lrPowerPV_1 := fbPV.arrDataSymo10[1].lrPowerAcInverter;
lrPowerPV_2 := fbPV.arrDataSymo10[2].lrPowerAcInverter;
lrPowerPV_3 := fbPV.arrDataSymo10[3].lrPowerAcInverter;
lrPowerPV_4 := fbPV.arrDataSymo10[4].lrPowerAcInverter;
lrPowerPV_5 := fbPV.arrDataSymo10[5].lrPowerAcInverter;
lrPowerPV_6 := fbPV.arrDataSymo10[6].lrPowerAcInverter;
lrPowerPV_7 := fbPV.arrDataSymo10[7].lrPowerAcInverter;
lrPowerPV_8 := fbPV.arrDataSymo10[8].lrPowerAcInverter;

(*
fbPV_2.arrUnitID_Inverter[1] := 7;
fbPV_2.arrUnitID_Inverter[2] := 8;

fbPV_2(
	bEnable:= TRUE, 
	sIPAdress:= '192.168.10.4', 
	arrUnitID_Inverter:= , 
	arrDataSymo10=> , 
	stDataEMPower_PV=> , 
	stDataEMCounter_PV=> , 
	diNrOfEM_OUT_PV=> );

lrPowerPV_7 := fbPV_2.arrDataSymo10[1].lrPowerAcInverter;
lrPowerPV_8 := fbPV_2.arrDataSymo10[2].lrPowerAcInverter;

*)
	
fbPVInt(
	bEnable:= TRUE, 
	bPowerDataInvers:= , 
	diNrOfEM_IN_PV:= fbPV.diNrOfEM_OUT_PV, 
	stDataPv=> , 
	diNrOfPv_OUT=> );
	
lrPowerPV := lrPowerPV_1 + lrPowerPV_2 + lrPowerPV_3 + lrPowerPV_4 + lrPowerPV_5 + lrPowerPV_6 + lrPowerPV_7 + lrPowerPV_8;
byErrorWarningPV := fbPVInt.stDataPv.byErrorWarning;

// EnergyCounter
fbPVCounter(
	byActiveTariff:= 1, 
	lrPowerInput:= 0 - lrPowerPV, 
	lrTotalCounterEnergy_Consumption=> , 
	lrTotalCounterEnergy_Production=> , 
	lrCounterEnergyT1_Consumption=> , 
	lrCounterEnergyT2_Consumption=> , 
	lrCounterEnergyT1_Production=> , 
	lrCounterEnergyT2_Production=> );
	
IF fbPVCounter.lrTotalCounterEnergy_Production > lrCounterPV THEN  	
	lrCounterPV := fbPVCounter.lrTotalCounterEnergy_Production;
END_IF

END_PROGRAM

// ---- POUs/prgGrid.TcPOU
PROGRAM prgGrid
VAR PERSISTENT
	rSizeGridConn				: REAL;									//{#lynus.ag#()}
	lrCounterGridProd			: LREAL;								//{#lynus.ag#()}
	lrCounterGridCons			: LREAL;								//{#lynus.ag#()}
	lrCounterGridProd2			: LREAL;								//{#lynus.ag#()}
	lrCounterGridCons2			: LREAL;								//{#lynus.ag#()}
	r_kWh_PriceGridCons			: REAL;									//{#lynus.ag#()}
	r_kWh_PriceGridProd			: REAL;									//{#lynus.ag#()}
END_VAR
VAR
	fbGrid						: FB_Grid_Power;
	lrGridPower					: LREAL;								//{#lynus.ag#()}
	lrGridPower2				: LREAL;								//{#lynus.ag#()}
	lrGridPower2RealTime		: LREAL;								//{#lynus.ag#()}
	fbGridCounter				: FB_EnergyCounter;
	fbGrid2						: FB_Measurement_EL3413_v1;
END_VAR

fbGrid(
	bEnable:= TRUE, 
	diNrOfEMS_IN:= prgEMS.fbEMS.diNrOfEMS_OUT, 
	diNrOfEM_IN_Grid:= prgBattery.fbBattery.diNrOfEM_OUT_Grid, 
	rSizeGridConn:= rSizeGridConn, 
	stDataGrid=> , 
	diNrOfGrid_OUT=> );
	
lrGridPower := fbGrid.stDataGrid.lrPower;

// EnergyCounter
fbGridCounter(
	byActiveTariff:= 1, 
	lrPowerInput:= lrGridPower, 
	lrTotalCounterEnergy_Consumption=> , 
	lrTotalCounterEnergy_Production=> , 
	lrCounterEnergyT1_Consumption=> , 
	lrCounterEnergyT2_Consumption=> , 
	lrCounterEnergyT1_Production=> , 
	lrCounterEnergyT2_Production=> );
	
IF fbGridCounter.lrTotalCounterEnergy_Production > lrCounterGridProd THEN  	
	lrCounterGridProd := fbGridCounter.lrTotalCounterEnergy_Production;
END_IF

IF fbGridCounter.lrTotalCounterEnergy_Consumption > lrCounterGridCons THEN  	
	lrCounterGridCons := fbGridCounter.lrTotalCounterEnergy_Consumption;
END_IF

fbGrid2(
	bEnable:= true, 
	bInvers_CH1:= , 
	bInvers_CH2:= , 
	bInvers_CH3:= , 
	uiCurrentTransformerRatio:= 60, 
	stDataEMPower=> , 
	stDataEMCounter=> , 
	stDataEMPowerRealTime=> , 
	stDataEMCounterRealTime=> );
	
lrGridPower2 := fbGrid2.stDataEMPower.lrPowerTotal;
lrGridPower2RealTime := fbGrid2.stDataEMPowerRealTime.lrPowerTotal;
lrCounterGridProd2 := fbGrid2.stDataEMCounter.lrTotalCounterEnergy_Production;
lrCounterGridCons2 := fbGrid2.stDataEMCounter.lrTotalCounterEnergy_Consumption;

END_PROGRAM

// ---- FB/FB_Measurement_EL3413_v1.TcPOU
FUNCTION_BLOCK FB_Measurement_EL3413_v1
VAR_INPUT
	bEnable							: BOOL;											//Enable the function
 	bInvers_CH1						: BOOL;											//Invert the Output data from Channel 1 
	bInvers_CH2						: BOOL;											//Invert the Output data from Channel 2 
	bInvers_CH3						: BOOL;											//Invert the Output data from Channel 3
	uiCurrentTransformerRatio		: UINT;											//Current Transformer Ratio  
END_VAR
VAR_OUTPUT
	stDataEMPower					: ST_ElectricMeter_Output_Power;				//Output structure with Data from Electric Meter (Power Data) 
	stDataEMCounter					: ST_ElectricMeter_Output_Counter;				//Output structure with Data from Electric Meter (Counter Data) 
	stDataEMPowerRealTime			: ST_ElectricMeter_Output_Power;				//Output structure with Data from Electric Meter (Power Data RealTime)
	stDataEMCounterRealTime			: ST_ElectricMeter_Output_Counter;				//Output structure with Data from Electric Meter (Counter Data RealTime) 
	diNrOfEM_OUT					: DINT;											//Active Number from the Electric Meter for using on other functions

END_VAR
VAR
	structEL3413_IO : MDP5001_340_341_8D4302F4;
	timDissableFunctions			: TON;											//Timer to dissable the Function after Lynus_Standards.Constants_General.tTimeDissableLynusFunctions Days without connection to the Lynus Cloud
	timResetConnectionOnGVL			: TON;											//Timer to try reset the connection Flag on the GVL. (When somebody delete the Connection Function and make only a onlinechange)
	timSetCounterValues				: TON;											//Timer to set the counter values from the KL3403 Function to the EM Function
	real_Multiplier_CH1: REAL;
	real_Multiplier_CH2: REAL;
	real_Multiplier_CH3: REAL;
	fbEM							: FB_ElectricMeter;								//Electric Meter Function
	fbEnergyCounter					: FB_EnergyCounter;								//FB energy Counter, because the KL3403 has no nice logic for the Energy value
	fbNumberDevice					: FB_NumberOfDevice;							//Function block to calcualte the number of the Device
	iStateGVLData					: INT;											//State machine to handle the data on the GVL

	

	real_CT_sec1: REAL;
	real_f1_Hz: REAL;
	real_f2_Hz: REAL;
	real_f3_Hz: REAL;
	lreal_S_VA_L1: LREAL;
	lreal_S_VA_L2: LREAL;
	lreal_S_VA_L3: LREAL;
	lreal_Q_var_L1: LREAL;
	lreal_Q_var_L2: LREAL;
	lreal_Q_var_L3: LREAL;
	lreal_E1_kWh: LREAL;
	lreal_E2_kWh: LREAL;
	lreal_E3_kWh: LREAL;
END_VAR

//Creator : Stefan Lackner
//Company : EfficientIO
//Date : xx.09.2023
//Version : 1.0.0.0


//With this function is possible to read out all Information from a EL3443

//NOTE for diNr.....Designation => 
//_IN = Here Data come in from other Functions or go out to other functions about the GVL
//_OUT = Here Data go out to other functions about the GVL

(*-------------------------------------------------------------Calcualte the number of EM---------------------------------------------------------------*)

fbNumberDevice(
	diActualNumberOfDevices:= Lynus_Standards.GVL_Energy.stNumberOfDevices.diNumberOfElectricMeters, 
	diMaxNumberOfDevices:= Constants_Energy.diMaxNumberOfElectricMeters, 
	udiCounterOnlineChange:= TwinCAT_SystemInfoVarList._AppInfo.OnlineChangeCnt, 
	bNumberIsCalculatet=> , 
	bFPNumberIsCalculatet=> , 
	bOnlineChange=> , 
	diNumberForThisDevice=> diNrOfEM_OUT, 
	diNumberOfTotalDevices=> );

//Write new Numer on GVL
IF fbNumberDevice.bFPNumberIsCalculatet THEN
	Lynus_Standards.GVL_Energy.stNumberOfDevices.diNumberOfElectricMeters := fbNumberDevice.diNumberOfTotalDevices;	
END_IF

//Delete old Number on GVL
IF fbNumberDevice.bOnlineChange THEN 
	Lynus_Standards.GVL_Energy.stNumberOfDevices.diNumberOfElectricMeters := diNrOfEM_OUT;	
		iStateGVLData := 1; 
END_IF

(*-------------------------------------------------------------Service from Backend is ready and check the connection to backen for dissabel/enable Function---------------------------------------------------------------*)

//Try to reset the variable for connection on the GVL. When all is normal then the Lynus Mqtt connection function set this variable to true in the next cycle
//When we have no connection to the backend then after Lynus_Standards.Constants_General.tTimeDissableLynusFunctions days the Function is dissabled with all of his functionalities
timResetConnectionOnGVL(IN:= NOT timResetConnectionOnGVL.Q, PT:= T#1H, Q=> , ET=> );
IF timResetConnectionOnGVL.Q THEN 
	Lynus_Standards.GVL_Communicator.bStateConnectionToEnableFunctions := FALSE; 
END_IF
IF NOT Lynus_Standards.GVL_Communicator.bStateConnectionToEnableFunctions THEN 
	timDissableFunctions.IN := TRUE; 
ELSE 
	timDissableFunctions.IN := FALSE; 
END_IF  
timDissableFunctions(IN:= , PT:= Lynus_Standards.Constants_General.tTimeDissableLynusFunctions, Q=> , ET=> );

// limit inputs
uiCurrentTransformerRatio	 := LIMIT (1,uiCurrentTransformerRatio,10000);

//Invert the Output data, because it is possible that the current transformers have been mounted in different mounting positions.
IF NOT bInvers_CH1 THEN
	real_Multiplier_CH1 := 1;
ELSE
	real_Multiplier_CH1 := -1;
END_IF
IF NOT bInvers_CH2 THEN
	real_Multiplier_CH2 := 1;
ELSE
	real_Multiplier_CH2 := -1;
END_IF
IF NOT bInvers_CH3 THEN
	real_Multiplier_CH3 := 1;
ELSE
	real_Multiplier_CH3 := -1;
END_IF


//Function
fbEM(
	bEnable:= bEnable AND NOT timDissableFunctions.Q, 
	bError:= , 
	bEnableReadOutFunction:= FALSE, 
	bWriteWithDelay:= TRUE, 
	bPowerDataInvers:= FALSE,
	bReadOutDataDone:= timSetCounterValues.Q,
	iTimeReadOutInterval:= 0, 
	iErrorCode:= , 
	iWarningCode:= , 
	lrTotalCounterEnergy_Consumption:= fbEnergyCounter.lrTotalCounterEnergy_Consumption,
	lrTotalCounterEnergy_Production:= fbEnergyCounter.lrTotalCounterEnergy_Production, 
	lrCounterEnergyT1_Consumption:= fbEnergyCounter.lrCounterEnergyT1_Consumption,
	lrCounterEnergyT2_Consumption:= fbEnergyCounter.lrCounterEnergyT2_Consumption,
	lrCounterEnergyT1_Production:= fbEnergyCounter.lrCounterEnergyT1_Production, 
	lrCounterEnergyT2_Production:= fbEnergyCounter.lrCounterEnergyT2_Production, 
	lrCurrentL1:=  DINT_TO_LREAL(structEL3413_IO.MDP5001_340_341_Input.MDP5001_340_PM_Inputs_Channel_1_Current)/1000000 * uiCurrentTransformerRatio,
	lrVoltageL1N:= DINT_TO_LREAL(structEL3413_IO.MDP5001_340_341_Input.MDP5001_340_PM_Inputs_Channel_1_Voltage)/10000,
	lrVoltageL1L2:= fbEM.lrVoltageL1N * 1.73, 
	lrPowerL1:=  DINT_TO_LREAL(structEL3413_IO.MDP5001_340_341_Input.MDP5001_340_PM_Inputs_Channel_1_Active_power)/100 * uiCurrentTransformerRatio * real_Multiplier_CH1, 
	lrCurrentL2:=  DINT_TO_LREAL(structEL3413_IO.MDP5001_340_341_Input.MDP5001_340_PM_Inputs_Channel_2_Current)/1000000 * uiCurrentTransformerRatio,
	lrVoltageL2N:= DINT_TO_LREAL(structEL3413_IO.MDP5001_340_341_Input.MDP5001_340_PM_Inputs_Channel_2_Voltage)/10000,
	lrVoltageL2L3:= fbEM.lrVoltageL2N * 1.73,
	lrPowerL2:= DINT_TO_LREAL(structEL3413_IO.MDP5001_340_341_Input.MDP5001_340_PM_Inputs_Channel_2_Active_power)/100 * uiCurrentTransformerRatio * real_Multiplier_CH2,
	lrCurrentL3:=  DINT_TO_LREAL(structEL3413_IO.MDP5001_340_341_Input.MDP5001_340_PM_Inputs_Channel_3_Current)/1000000 * uiCurrentTransformerRatio,
	lrVoltageL3N:= DINT_TO_LREAL(structEL3413_IO.MDP5001_340_341_Input.MDP5001_340_PM_Inputs_Channel_3_Voltage)/10000,
	lrVoltageL3L1:= fbEM.lrVoltageL3N * 1.73,
	lrPowerL3:= DINT_TO_LREAL(structEL3413_IO.MDP5001_340_341_Input.MDP5001_340_PM_Inputs_Channel_3_Active_power)/100 * uiCurrentTransformerRatio * real_Multiplier_CH3,
	lrPowerTotal:= fbEM.lrPowerL1+fbEM.lrPowerL2+fbEM.lrPowerL3,
 	lrFrequency:= (real_f1_Hz + real_f2_Hz + real_f3_Hz)/3 , 
 	lrApparentPowerTotal:= (lreal_S_VA_L1 + lreal_S_VA_L2 + lreal_S_VA_L3),
	lrReactivePowerTotal:= (lreal_Q_var_L1 +lreal_Q_var_L2 + lreal_Q_var_L3), 
	tTimDelayOutput:= T#5S, 
	stDataEMOutPower=> stDataEMPowerRealTime, 
	stDataEMOutPowerDelay=> stDataEMPower, 
	stDataEMOutCounter=> stDataEMCounterRealTime,
	stDataEMOutCounterDelay=> stDataEMCounter,
	bReadOutMeter=> );
(*----------------------------------------------------------------------------------------Energy Counter Function----------------------------------------------------------------------------------------------*)

fbEnergyCounter(
	byActiveTariff:= 1, 
	lrPowerInput:= (fbEM.lrPowerTotal) / 1000, 
	lrTotalCounterEnergy_Consumption=> , 
	lrTotalCounterEnergy_Production=> , 
	lrCounterEnergyT1_Consumption=> , 
	lrCounterEnergyT2_Consumption=> , 
	lrCounterEnergyT1_Production=> , 
	lrCounterEnergyT2_Production=> );


IF (fbEM.lrPowerL1 * fbEM.lrPowerL1 + lreal_Q_var_L1 * lreal_Q_var_L1) <> 0 THEN 
	lreal_S_VA_L1:=SQRT(fbEM.lrPowerL1 * fbEM.lrPowerL1 + lreal_Q_var_L1 * lreal_Q_var_L1);
END_IF
IF (fbEM.lrPowerL2 * fbEM.lrPowerL2 + lreal_Q_var_L2 * lreal_Q_var_L2) <> 0 THEN 
	lreal_S_VA_L2:=SQRT(fbEM.lrPowerL2 * fbEM.lrPowerL2 + lreal_Q_var_L2 * lreal_Q_var_L2);
END_IF
IF (fbEM.lrPowerL3 * fbEM.lrPowerL3 + lreal_Q_var_L3 * lreal_Q_var_L3) <> 0 THEN 
	lreal_S_VA_L3:=SQRT(fbEM.lrPowerL3 * fbEM.lrPowerL3 + lreal_Q_var_L3 * lreal_Q_var_L3);
END_IF

CASE  structEL3413_IO.MDP5001_340_341_Input.MDP5001_340_PM_Inputs_Channel_1_Index OF
	1: (* Q *)
		lreal_Q_var_L1 :=DINT_TO_LREAL(structEL3413_IO.MDP5001_340_341_Input.MDP5001_340_PM_Inputs_Channel_1_Variant_value)/100 * uiCurrentTransformerRatio;
		structEL3413_IO.MDP5001_340_341_Output.MDP5001_340_PM_Outputs_Channel_1_Index := 2;
	2: (* E *)
		lreal_E1_kWh := DINT_TO_LREAL(structEL3413_IO.MDP5001_340_341_Input.MDP5001_340_PM_Inputs_Channel_1_Variant_value )/1000000 * uiCurrentTransformerRatio;
		structEL3413_IO.MDP5001_340_341_Output.MDP5001_340_PM_Outputs_Channel_1_Index := 4;
	4: (* f *)
		real_f1_Hz:=DINT_TO_REAL(structEL3413_IO.MDP5001_340_341_Input.MDP5001_340_PM_Inputs_Channel_1_Variant_value )/10;
		structEL3413_IO.MDP5001_340_341_Output.MDP5001_340_PM_Outputs_Channel_1_Index := 1;
ELSE
		structEL3413_IO.MDP5001_340_341_Output.MDP5001_340_PM_Outputs_Channel_1_Index := 1;
END_CASE
CASE  structEL3413_IO.MDP5001_340_341_Input.MDP5001_340_PM_Inputs_Channel_2_Index OF
	1: (* Q *)
		lreal_Q_var_L2 :=DINT_TO_LREAL(structEL3413_IO.MDP5001_340_341_Input.MDP5001_340_PM_Inputs_Channel_2_Variant_value)/100 * uiCurrentTransformerRatio;
		structEL3413_IO.MDP5001_340_341_Output.MDP5001_340_PM_Outputs_Channel_2_Index := 2;
	2: (* E *)
		lreal_E2_kWh := DINT_TO_LREAL(structEL3413_IO.MDP5001_340_341_Input.MDP5001_340_PM_Inputs_Channel_2_Variant_value )/1000000 * uiCurrentTransformerRatio;
		structEL3413_IO.MDP5001_340_341_Output.MDP5001_340_PM_Outputs_Channel_2_Index := 4;
	4: (* f *)
		real_f2_Hz:=DINT_TO_REAL(structEL3413_IO.MDP5001_340_341_Input.MDP5001_340_PM_Inputs_Channel_2_Variant_value )/10;
		structEL3413_IO.MDP5001_340_341_Output.MDP5001_340_PM_Outputs_Channel_2_Index := 1;
ELSE
		structEL3413_IO.MDP5001_340_341_Output.MDP5001_340_PM_Outputs_Channel_2_Index := 1;
END_CASE
CASE  structEL3413_IO.MDP5001_340_341_Input.MDP5001_340_PM_Inputs_Channel_3_Index OF
	1: (* Q *)
		lreal_Q_var_L3 :=DINT_TO_LREAL(structEL3413_IO.MDP5001_340_341_Input.MDP5001_340_PM_Inputs_Channel_3_Variant_value)/100 * uiCurrentTransformerRatio;
		structEL3413_IO.MDP5001_340_341_Output.MDP5001_340_PM_Outputs_Channel_3_Index := 2;
	2: (* E *)
		lreal_E3_kWh := DINT_TO_LREAL(structEL3413_IO.MDP5001_340_341_Input.MDP5001_340_PM_Inputs_Channel_3_Variant_value )/1000000 * uiCurrentTransformerRatio;
		structEL3413_IO.MDP5001_340_341_Output.MDP5001_340_PM_Outputs_Channel_3_Index := 4;
	4: (* f *)
		real_f3_Hz:=DINT_TO_REAL(structEL3413_IO.MDP5001_340_341_Input.MDP5001_340_PM_Inputs_Channel_3_Variant_value )/10;
		structEL3413_IO.MDP5001_340_341_Output.MDP5001_340_PM_Outputs_Channel_3_Index := 1;
ELSE
		structEL3413_IO.MDP5001_340_341_Output.MDP5001_340_PM_Outputs_Channel_3_Index := 1;
END_CASE


IF IsFinite(F_LREAL(fbEnergyCounter.lrTotalCounterEnergy_Production)) THEN stDataEMCounter.lrTotalCounterEnergy_Production := LINT_TO_LREAL(LREAL_TO_LINT(fbEnergyCounter.lrTotalCounterEnergy_Production * 100)) / 100; END_IF
IF IsFinite(F_LREAL(fbEnergyCounter.lrTotalCounterEnergy_Consumption)) THEN stDataEMCounter.lrTotalCounterEnergy_Consumption := LINT_TO_LREAL(LREAL_TO_LINT(fbEnergyCounter.lrTotalCounterEnergy_Consumption * 100)) / 100; END_IF

END_FUNCTION_BLOCK

// ---- POUs/prgCS.TcPOU
PROGRAM prgCS
VAR PERSISTENT
	bEnabledCS				: BOOL;									//{#lynus.ag#()}
	byPrioCS				: BYTE;									//{#lynus.ag#()}
	bySOC_E_CS				: BYTE;									//{#lynus.ag#()}
	bySOC_D_CS				: BYTE;									//{#lynus.ag#()}
	byMinPowerCS			: BYTE;									//{#lynus.ag#()}
	rMaxPowerCS				: REAL;									//{#lynus.ag#()}
	lrCounterCS				: LREAL;								//{#lynus.ag#()}
	bManualyOn				: BOOL;									//{#lynus.ag#()}
	byMinPower				: BYTE;									//{#lynus.ag#()}
	byManualyTargetPower	: BYTE;									//{#lynus.ag#()}
	m_ChargingLimit			: BOOL;									//{#lynus.ag#()}
	bOnEmergPowerOff		: BOOL;									//{#lynus.ag#()}
END_VAR
VAR
	fbCS					: FB_ECS_Alpitronic_Hypercharger_1;
	fbCSCounter				: FB_EnergyCounter;
	bIsEnabledCS			: BOOL;									//{#lynus.ag#()}
	byErrorWarningCS		: BYTE;									//{#lynus.ag#()}
	byStateMinPowerCS		: BYTE;									//{#lynus.ag#()}
	rTargetPowerCS			: REAL;									//{#lynus.ag#()}
	bCarConnected			: BOOL;									//{#lynus.ag#()}
	rChrgTime				: REAL;									//{#lynus.ag#()}
	lrPowerCS				: LREAL;								//{#lynus.ag#()}
	bSManualyOn				: BOOL;									//{#lynus.ag#()}
	bySManualyTargetPower	: BYTE;									//{#lynus.ag#()}
	str_IP: STRING(15):='192.168.10.10';
	rSOC_1					: REAL;									//{#lynus.ag#()}
	rSOC_2					: REAL;									//{#lynus.ag#()}
	f_Trig_CarConntected: f_trig;
	bSOnEmergPowerOff		: BOOL;									//{#lynus.ag#()}
END_VAR

fbCS.stSetupECS.byDisableSOC := bySOC_D_CS;
fbCS.stSetupECS.byEnableSOC := bySOC_E_CS;
fbCS.stSetupECS.byPriority := byPrioCS;
fbCS.stSetupECS.rMaxPower := rMaxPowerCS;
fbCS.stSetupECS.byCSMinPower := byMinPowerCS;
fbCS.stSetupECS.bManualyOn := bManualyOn;
fbCS.stSetupECS.byManualyTargetPower := byManualyTargetPower;
fbCS.stSetupECS.byCSMinPower := byMinPower;
fbCS.stSetupECS.bOnEmergPowerOff := bOnEmergPowerOff;


// Kofler special requirement for allowing to charge with maximium power and not PV surplus
// no battery used for charging the car. Battery Prio 2, CS prio 1
f_Trig_CarConntected(Clk := bCarConnected);
IF f_Trig_CarConntected.Q THEN 
	m_ChargingLimit := TRUE;
END_IF

IF m_ChargingLimit THEN
	fbCS.stSetupECS.byCSMinPower := byMinPowerCS;
ELSE
	fbCS.stSetupECS.byCSMinPower := 100;
END_IF
	
fbCS(
	bEnable:= bEnabledCS, 
	bPowerDataInvers:= , 
	byUnitID:= 1,				//Allways 1 
	diNrOfEMS_IN:= prgEMS.fbEMS.diNrOfEMS_OUT, 
	diNrOfEM_IN_CS:= , 
	sIPAdress:= str_IP, 
	stSetupECS:= , 
	stDataECS=> , 
	diNrOfECS_OUT=> );

bIsEnabledCS := fbCS.stDataECS.bEnabled;
byStateMinPowerCS := fbCS.stDataECS.bySCSMinPower;
rTargetPowerCS := fbCS.stDataECS.rTargetPower;	
byErrorWarningCS := fbCS.stDataECS.byErrorWarning;
bCarConnected := fbCS.stDataECS.bCarConnected;
rChrgTime := MAX(fbCS.stDataECS.arrChargingTimeInMin[1],fbCS.stDataECS.arrChargingTimeInMin[2]);
lrPowerCS := fbCS.stDataECS.lrTotalPower;
bSManualyOn := fbCS.stDataECS.bSManualyOn;
bSOnEmergPowerOff := fbCS.stDataECS.bSOnEmergPowerOff;

bySManualyTargetPower := fbCS.stDataECS.bySManualyTargetPower;
rSOC_1	:= DWORD_TO_REAL(fbCS.stDataECS.arrSocketSOCCar[1]);
rSOC_2	:= DWORD_TO_REAL(fbCS.stDataECS.arrSocketSOCCar[2]);						

// EnergyCounter
fbCSCounter(
	byActiveTariff:= 1, 
	lrPowerInput:= lrPowerCS, 
	lrTotalCounterEnergy_Consumption=> );
	
IF fbCSCounter.lrTotalCounterEnergy_Consumption > lrCounterCS THEN  	
	lrCounterCS := fbCSCounter.lrTotalCounterEnergy_Consumption;
END_IF

END_PROGRAM

// ---- FB/FB_ECS_Alpitronic_Hypercharger_1.TcPOU
FUNCTION_BLOCK FB_ECS_Alpitronic_Hypercharger_1
VAR_INPUT PERSISTENT
	bEnable										: BOOL;																			//{#lynus.ag#()} //Enable the Fuctionblock and his logic
	bPowerDataInvers							: BOOL;																			//With True its possible to invert all received power data from the electric meter
	byElectricFuseLine							: BYTE; 																		//Electric Fuse Line on wich the ECS is connected => 1 2 3 (If 0 then this charging station is not connected to a Electric Fuse Line)
	byUnitID									: BYTE;																			//Unit ID 
	diNrOfEMS_IN								: DINT;																			//Number of EMS what control this Device.
	diNrOfEM_IN_CS								: DINT;																			//Number of the electric meter for incoming power data. (Power Data for this Device)
	sIPAdress									: STRING(15);																	//IP Adress from the Alfen charging station
	stSetupECS									: ST_Setup_ECS;																	//{#lynus.ag#()} //Setup charging station
END_VAR
VAR_OUTPUT
	stDataECS									: ST_ECS_Output;																//{#lynus.ag#()} //Electric charging station output data
	diNrOfECS_OUT								: DINT;																			//Active Number from the Electric charging Function for using on other functions
	lrTotalPowerECSRealTime						: LREAL;																		//Total Electric Power in kW read out directly from the Charging station. (Real time)
END_VAR
VAR
	fbCS										: FB_ElectricChargingStation_1;													//Function block for electric charging station
	fbNumberDevice								: FB_NumberOfDevice;															//Function block to calcualte the number of the Device
	fbDIExternalLock							: FB_XL1XXX_DI;																	//Digital Input from external loock signal
	fbMBRead_FC4								: FB_MBReadInputRegs ;															//Modbus Read Function (FC4)
	fbMBWrite_FC16								: FB_MBWriteRegs;																//Modbus Write Function (FC16)
	fbConvertDwordToWord						: FB_CV_DWORD_TO_WORD;															//Convert Dword to Word
	fbConvertWordToDord							: FB_CV_WORD_TO_DWORD;															//Convert Word to Dword
	timDelay									: TON;																			//Timer for Delay between Requests
	timTimeout									: TON;																			//Timer for Timeout
	timDissableFunctions						: TON;																			//Timer to dissable the Function after Lynus_Standards.Constants_General.tTimeDissableLynusFunctions Days without connection to the Lynus Cloud
	timResetConnectionOnGVL						: TON;																			//Timer to try reset the connection Flag on the GVL. (When somebody delete the Connection Function and make only a onlinechange)
	timDelayStart								: TON;																			//Timer to start the state machine with Daley after enabling or after the system ist restartet
	FPError_FC_4								: R_TRIG;																		//Internal positive Edge
	FPError_FC_16								: R_TRIG;																		//Internal positive Edge
	FPEnable									: R_TRIG;																		//Internal positive Edge
	arrPD										: ARRAY[1..15] OF FB_PersistentData_Number;										//Function to save persistent data
	arrEnergyCounterSocket						: ARRAY[1..4] OF FB_EnergyCounter;												//FB energy Counter, because the charging station not deliver the total energy Counter in kWh
	fbPDString									: FB_PersistentData_String;														//Function to save persistent string data
	arrBuffer_FC4								: ARRAY[1..9] OF WORD;															//Buffer with Data from FC3
	arrBuffer_FC16								: ARRAY[1..2] OF WORD;															//Buffer with Data from FC16
	arrConnectorState							: ARRAY[1..4] OF WORD;															//Connector State
	arrChargingTime								: ARRAY[1..4] OF WORD;															//Charging Time in seconds
	arrSOCCar									: ARRAY[1..4] OF WORD;															//SOC from the Car
	arrPowerConnector							: ARRAY[1..4] OF DWORD;															//Power in W from each Connector
	arrEnergySession							: ARRAY[1..4] OF REAL;															//Energy Session in kWh
	bErrorCS									: BOOL;																			//Error State from the charging station
	bMBTCPError									: BOOL;																			//Modbus TCP Function Error																	
	byWaitInStep								: BYTE;																			//Wait in Step before start to clean data on PLC
	iStateGVLData								: INT;																			//State machine to handle the data on the GVL
	iStateModbusRead							: INT;																			//State machine for read out Data over Modbus RTU
	iStateModbusWrite							: INT;																			//State machine for write Data over Modbus RTU
	iStateModbusError							: INT;																			//State machine for error out Data over Modbus RTU	
	iStateModbus_CP								: INT;																			//Variable to compare the state machine variable to set or reset the timeout timer
	wNumberOfConnectors							: WORD;																			//Number of real connecotrs on the charging station
	wStationState								: WORD;																			//Charging Station State
	wConnectorInProgress						: WORD;																			//Shows the Connector in Progress when we have more then 1 Connector	
	diNumberOfActiveBatterys					: DINT;																			//Number of active batterys
	diNumberOfBatteryInverterInEPO				: DINT;																			//Number of battery inverters that work in Emergency Power operation 
	diLPForGVL									: DINT;																			//Loop to clean old data on GVL
	diCounterForGVL								: DINT;																			//Counter to clean old data on GVL
	dwSumSOC									: DWORD;																		//Sum of the SOC from all batterys
	dwTargetPower								: DWORD;																		//Target Power in Watt to send to the charging station
	liLPBatteryData								: LINT;																			//Loop to check some data from batterys
	liLPInEPO									: LINT;																			//Loop to check if 1 or more battery inverters build a island grid
	mtest: BOOL;

END_VAR
VAR PERSISTENT
	diNrOfEMS_IN_CP								: DINT;																			//Number of EMS what control this Device to compare with the original
END_VAR

//Creator : Kai Ebensperger
//Company : Lynus AG
//Date : 07.10.2021
//Version : 1.0.0.0

//With this Funcition its possible to communicate with a Alpitronic Hypercharger charging station over Modbus TCP.
//Its possible to controll the charging station over the charge power with the unit W
//This Charging station is a DC Hypercharger System.
//This API deliver the real Number of Connectors on the charging station
//To switch off the charging station send 0 Power to the charging station
//The minimal Curretn is set to 7.5 Ampere on AC site, bacause with al values that are < 5kW its not possible to charge the Car on DC site
//This Function Block support maximal 4 Connectors

//Versions that are supported : 1.3A Date : October 2020

//NOTE for diNr.....Designation => 
//_IN = Here Data come in from other Functions or go out to other functions about the GVL
//_OUT = Here Data go out to other functions about the GVL

(*--------------------------------------------------------------------------------------------Limits-------------------------------------------------------------------------------------*)

diNrOfEMS_IN := LIMIT(0,diNrOfEMS_IN,Constants_Energy.diMaxNumberOfEMS);
	diNrOfEM_IN_CS := LIMIT(0,diNrOfEM_IN_CS,Constants_Energy.diMaxNumberOfElectricMeters);	

(*------------------------------------------------------------------Power Data----------------------------------------------------------------------------*)

//Energy Counter Functions
arrEnergyCounterSocket[1](
	byActiveTariff:= 1, 
	lrPowerInput:= DWORD_TO_REAL(arrPowerConnector[1]) / 1000, 
	lrTotalCounterEnergy_Consumption=> , 
	lrTotalCounterEnergy_Production=> , 
	lrCounterEnergyT1_Consumption=> , 
	lrCounterEnergyT2_Consumption=> , 
	lrCounterEnergyT1_Production=> , 
	lrCounterEnergyT2_Production=> );
	
arrEnergyCounterSocket[2](
	byActiveTariff:= 1, 
	lrPowerInput:= DWORD_TO_REAL(arrPowerConnector[2]) / 1000, 
	lrTotalCounterEnergy_Consumption=> , 
	lrTotalCounterEnergy_Production=> , 
	lrCounterEnergyT1_Consumption=> , 
	lrCounterEnergyT2_Consumption=> , 
	lrCounterEnergyT1_Production=> , 
	lrCounterEnergyT2_Production=> );

arrEnergyCounterSocket[3](
	byActiveTariff:= 1, 
	lrPowerInput:= DWORD_TO_REAL(arrPowerConnector[3]) / 1000, 
	lrTotalCounterEnergy_Consumption=> , 
	lrTotalCounterEnergy_Production=> , 
	lrCounterEnergyT1_Consumption=> , 
	lrCounterEnergyT2_Consumption=> , 
	lrCounterEnergyT1_Production=> , 
	lrCounterEnergyT2_Production=> );	
	
arrEnergyCounterSocket[4](
	byActiveTariff:= 1, 
	lrPowerInput:= DWORD_TO_REAL(arrPowerConnector[4]) / 1000, 
	lrTotalCounterEnergy_Consumption=> , 
	lrTotalCounterEnergy_Production=> , 
	lrCounterEnergyT1_Consumption=> , 
	lrCounterEnergyT2_Consumption=> , 
	lrCounterEnergyT1_Production=> , 
	lrCounterEnergyT2_Production=> );

IF diNrOfEM_IN_CS <> 0 THEN
	//Energy Session Input data
	fbCS.bCalculateEnergySession := FALSE;
	fbCS.arrSocketPowerECS[1] := 0;
	fbCS.arrSocketPowerECS[2] := 0;
	fbCS.arrSocketPowerECS[3] := 0;
	fbCS.arrSocketPowerECS[4] := 0;
	fbCS.arrSocketEnergySession[1] := 0;
	fbCS.arrSocketEnergySession[2] := 0;
	fbCS.arrSocketEnergySession[3] := 0;
	fbCS.arrSocketEnergySession[4] := 0;
		IF NOT bPowerDataInvers THEN
			//Energy meter input data for cs Function block
			fbCS.lrCounterEnergyT1_Consumption := Lynus_Standards.GVL_Energy.stDataElectricMeters[diNrOfEM_IN_CS].lrCounterEnergyT1_Production * 1000;
			fbCS.lrCounterEnergyT2_Consumption := Lynus_Standards.GVL_Energy.stDataElectricMeters[diNrOfEM_IN_CS].lrCounterEnergyT2_Production * 1000;
			fbCS.lrCounterEnergyT1_Production := Lynus_Standards.GVL_Energy.stDataElectricMeters[diNrOfEM_IN_CS].lrCounterEnergyT1_Consumption * 1000;
			fbCS.lrCounterEnergyT2_Production := Lynus_Standards.GVL_Energy.stDataElectricMeters[diNrOfEM_IN_CS].lrCounterEnergyT1_Consumption * 1000;
			fbCS.lrTotalCounterEnergy_Consumption := Lynus_Standards.GVL_Energy.stDataElectricMeters[diNrOfEM_IN_CS].lrTotalCounterEnergy_Production * 1000;
			fbCS.lrTotalCounterEnergy_Production := Lynus_Standards.GVL_Energy.stDataElectricMeters[diNrOfEM_IN_CS].lrTotalCounterEnergy_Consumption * 1000;
				fbCS.lrTotalPowerECS := (Lynus_Standards.GVL_Energy.stDataElectricMeters[diNrOfEM_IN_CS].lrPower * 1000) * - 1;
		ELSE
			//Energy meter input data for cs Function block
			fbCS.lrCounterEnergyT1_Consumption := Lynus_Standards.GVL_Energy.stDataElectricMeters[diNrOfEM_IN_CS].lrCounterEnergyT1_Consumption * 1000;
			fbCS.lrCounterEnergyT2_Consumption := Lynus_Standards.GVL_Energy.stDataElectricMeters[diNrOfEM_IN_CS].lrCounterEnergyT2_Consumption * 1000;
			fbCS.lrCounterEnergyT1_Production := Lynus_Standards.GVL_Energy.stDataElectricMeters[diNrOfEM_IN_CS].lrCounterEnergyT1_Production * 1000;
			fbCS.lrCounterEnergyT2_Production := Lynus_Standards.GVL_Energy.stDataElectricMeters[diNrOfEM_IN_CS].lrCounterEnergyT2_Production * 1000;
			fbCS.lrTotalCounterEnergy_Consumption := Lynus_Standards.GVL_Energy.stDataElectricMeters[diNrOfEM_IN_CS].lrTotalCounterEnergy_Consumption * 1000;
			fbCS.lrTotalCounterEnergy_Production := Lynus_Standards.GVL_Energy.stDataElectricMeters[diNrOfEM_IN_CS].lrTotalCounterEnergy_Production * 1000;
				fbCS.lrTotalPowerECS := Lynus_Standards.GVL_Energy.stDataElectricMeters[diNrOfEM_IN_CS].lrPower * 1000;
		END_IF
ELSE
	//Energy meter input data for cs Function block
	fbCS.lrCounterEnergyT1_Consumption := arrEnergyCounterSocket[1].lrCounterEnergyT1_Consumption + arrEnergyCounterSocket[2].lrCounterEnergyT1_Consumption + arrEnergyCounterSocket[3].lrCounterEnergyT1_Consumption + arrEnergyCounterSocket[4].lrCounterEnergyT1_Consumption;
	fbCS.lrCounterEnergyT1_Consumption := fbCS.lrCounterEnergyT1_Consumption * 1000;
	fbCS.lrCounterEnergyT2_Consumption := arrEnergyCounterSocket[1].lrCounterEnergyT2_Consumption + arrEnergyCounterSocket[2].lrCounterEnergyT2_Consumption + arrEnergyCounterSocket[3].lrCounterEnergyT2_Consumption + arrEnergyCounterSocket[4].lrCounterEnergyT2_Consumption;
	fbCS.lrCounterEnergyT2_Consumption := fbCS.lrCounterEnergyT2_Consumption * 1000;
	fbCS.lrCounterEnergyT1_Production := arrEnergyCounterSocket[1].lrCounterEnergyT1_Production + arrEnergyCounterSocket[2].lrCounterEnergyT1_Production + arrEnergyCounterSocket[3].lrCounterEnergyT1_Production + arrEnergyCounterSocket[4].lrCounterEnergyT1_Production;
	fbCS.lrCounterEnergyT1_Production := fbCS.lrCounterEnergyT1_Production * 1000;
	fbCS.lrCounterEnergyT2_Production := arrEnergyCounterSocket[1].lrCounterEnergyT2_Production + arrEnergyCounterSocket[2].lrCounterEnergyT2_Production + arrEnergyCounterSocket[3].lrCounterEnergyT2_Production + arrEnergyCounterSocket[4].lrCounterEnergyT2_Production;
	fbCS.lrCounterEnergyT2_Production := fbCS.lrCounterEnergyT2_Production * 1000;
	fbCS.lrTotalCounterEnergy_Consumption := fbCS.lrCounterEnergyT1_Consumption + fbCS.lrCounterEnergyT2_Consumption;
	fbCS.lrTotalCounterEnergy_Production := fbCS.lrCounterEnergyT1_Production + fbCS.lrCounterEnergyT2_Production;
		fbCS.lrTotalPowerECS := arrPowerConnector[1] + arrPowerConnector[2] + arrPowerConnector[3] + arrPowerConnector[4];
	//Energy Session Input data
	fbCS.bCalculateEnergySession := FALSE;
	fbCS.arrSocketPowerECS[1] := arrPowerConnector[1];
	fbCS.arrSocketPowerECS[2] := arrPowerConnector[2];
	fbCS.arrSocketPowerECS[3] := arrPowerConnector[3];
	fbCS.arrSocketPowerECS[4] := arrPowerConnector[4];
	fbCS.arrSocketEnergySession[1] := arrEnergySession[1] * 1000;
	fbCS.arrSocketEnergySession[2] := arrEnergySession[2] * 1000;
	fbCS.arrSocketEnergySession[3] := arrEnergySession[3] * 1000;
	fbCS.arrSocketEnergySession[4] := arrEnergySession[4] * 1000;
END_IF			

(*-------------------------------------------------------------Calcualte the number of ECS---------------------------------------------------------------*)

fbNumberDevice(
	diActualNumberOfDevices:= Lynus_Standards.GVL_Energy.stNumberOfDevices.diNumberOfECS, 
	diMaxNumberOfDevices:= Constants_Energy.diMaxNumberOfElectricChargingStations, 
	udiCounterOnlineChange:= TwinCAT_SystemInfoVarList._AppInfo.OnlineChangeCnt, 
	bNumberIsCalculatet=> , 
	bFPNumberIsCalculatet=> , 
	bOnlineChange=> , 
	diNumberForThisDevice=> diNrOfECS_OUT, 
	diNumberOfTotalDevices=> );

//Write new Numer on GVL
IF fbNumberDevice.bFPNumberIsCalculatet THEN
	Lynus_Standards.GVL_Energy.stNumberOfDevices.diNumberOfECS := fbNumberDevice.diNumberOfTotalDevices;	
END_IF 

//Delete old Number on GVL
IF fbNumberDevice.bOnlineChange THEN 
	Lynus_Standards.GVL_Energy.stNumberOfDevices.diNumberOfECS := diNrOfECS_OUT;	
		iStateGVLData := 1;
END_IF

(*-------------------------------------------------------------Service from Backend is ready and check the connection to backen for dissabel/enable Function---------------------------------------------------------------*)

//Try to reset the variable for connection on the GVL. When all is normal then the Lynus Mqtt connection function set this variable to true in the next cycle
//When we have no connection to the backend then after Lynus_Standards.Constants_General.tTimeDissableLynusFunctions days the Function is dissabled with all of his functionalities
timResetConnectionOnGVL(IN:= NOT timResetConnectionOnGVL.Q, PT:= T#1H, Q=> , ET=> );
	IF timResetConnectionOnGVL.Q THEN Lynus_Standards.GVL_Communicator.bStateConnectionToEnableFunctions := FALSE; END_IF
		IF NOT Lynus_Standards.GVL_Communicator.bStateConnectionToEnableFunctions THEN timDissableFunctions.IN := TRUE; ELSE timDissableFunctions.IN := FALSE; END_IF  
			timDissableFunctions(IN:= , PT:= Lynus_Standards.Constants_General.tTimeDissableLynusFunctions, Q=> , ET=> );
			
(*--------------------------------------------------------------------------------------------State Machine Read--------------------------------------------------------------------------------------*)

//Timer for Delay
timDelay(IN:= , PT:= T#250MS, Q=> , ET=> );

//Timer for Timeout in Statemachine
IF (iStateModbusRead > 0 AND iStateModbusRead <= 3 AND iStateModbusRead = iStateModbus_CP) OR
		(iStateModbusWrite > 0 AND iStateModbusWrite <= 1 AND iStateModbusWrite = iStateModbus_CP) THEN
			timTimeout.IN := TRUE;
ELSE	
			timTimeout.IN := FALSE;
END_IF 
	//Timeout Timer is dissabled when the Init Step is aktiv or the function is not enabled
	IF (iStateModbusRead = 0 AND iStateModbusWrite = 0) OR NOT bEnable THEN timTimeout.IN := FALSE; END_IF
		timTimeout(IN:= , PT:= T#10S, Q=> , ET=> );

//Enable with Delay that not all sockets have to be created at the same time
timDelayStart(IN:= bEnable, PT:= T#20MS * diNrOfECS_OUT, Q=> , ET=> );
	FPEnable(CLK:= timDelayStart.Q, Q=> );

IF FPEnable.Q AND iStateModbusRead = 0 AND iStateModbusWrite = 0 THEN iStateModbusRead := 1; wConnectorInProgress := 1; END_IF		
		
//Not Enabled
IF NOT bEnable THEN iStateModbusRead := 0; iStateModbusError := 0; iStateModbusWrite := 0; END_IF		
		
CASE iStateModbusRead OF

	0://Init Step 
		iStateModbus_CP := 0;
			timDelay.IN := FALSE;
				fbMBRead_FC4.bExecute := FALSE;
					fbMBWrite_FC16.bExecute := FALSE;
						wConnectorInProgress := 0;
		arrConnectorState[1] := 0; arrConnectorState[2] := 0; arrConnectorState[3] := 0; arrConnectorState[4] := 0;
	
	1://Read Out the Number of connectors and the Charging station State (Register 2 and 3)
		iStateModbus_CP := iStateModbusRead;
		
		//Reset Write
		fbMBWrite_FC16.bExecute := FALSE;
			
		//Start Read
		fbMBRead_FC4.nQuantity := 2;
			fbMBRead_FC4.nMBAddr := 2;
				fbMBRead_FC4.bExecute := TRUE;
					fbMBRead_FC4.nUnitID := byUnitID;
			
		IF fbMBRead_FC4.bBusy THEN timDelay.IN := TRUE; END_IF
		
		//Wait for Delay, copy Data and then next step
		IF NOT fbMBRead_FC4.bBusy AND NOT fbMBRead_FC4.bError AND timDelay.Q THEN
			//Number of real Connectors
			wNumberOfConnectors := arrBuffer_FC4[1];
			//Charging station State
			wStationState := arrBuffer_FC4[2];	 
			//Connector in Progress
			wConnectorInProgress := LIMIT(1,wConnectorInProgress,4);
			//Go to Next Step
			fbMBRead_FC4.bExecute := FALSE;
				timDelay.IN := FALSE;		
					iStateModbusRead := 2;
		END_IF	

		//Error or Timeout
		IF FPError_FC_4.Q OR timTimeout.Q THEN
			iStateModbusError := 300;
		END_IF
		
	2://Read Out the Information of the real connecotrs (Register "1"00 to "1"08)
		iStateModbus_CP := iStateModbusRead;
		
		//Start Read
		fbMBRead_FC4.nQuantity := 9;
			fbMBRead_FC4.nMBAddr := 100 * wConnectorInProgress;
				fbMBRead_FC4.bExecute := TRUE;
					fbMBRead_FC4.nUnitID := byUnitID;
			
		IF fbMBRead_FC4.bBusy THEN timDelay.IN := TRUE; END_IF
		
		//Wait for Delay, copy Data and then next step
		IF NOT fbMBRead_FC4.bBusy AND NOT fbMBRead_FC4.bError AND timDelay.Q THEN
			//Connecotor State
			arrConnectorState[wConnectorInProgress] := arrBuffer_FC4[1];
			//Connector Power
			fbConvertWordToDord(wInputValue_1:= arrBuffer_FC4[5], wInputValue_2:= arrBuffer_FC4[6], eByteOrderForConvert:= eByteOrder.eBigEndian, dwOutputValue=> );
				arrPowerConnector[wConnectorInProgress] := fbConvertWordToDord.dwOutputValue;
			//Charging Time in Seconds
			arrChargingTime[wConnectorInProgress] := arrBuffer_FC4[7];
			//Energy Session
			arrEnergySession[wConnectorInProgress] := WORD_TO_REAL(arrBuffer_FC4[8]) / 100;
			//SOC from the Car
			arrSOCCar[wConnectorInProgress] := arrBuffer_FC4[9] / 100;
			//Go to Next Step
			fbMBRead_FC4.bExecute := FALSE;
				timDelay.IN := FALSE;		
					iStateModbusRead := 3;
		END_IF	

		//Error or Timeout
		IF FPError_FC_4.Q OR timTimeout.Q THEN
			iStateModbusError := 300;
		END_IF
		
	3://Wait 1 Step to reset the delay counter befor start to write
		iStateModbus_CP := iStateModbusRead;
		
			iStateModbusWrite := 1;
				//-1 because 0 is the Init Step for Read
				iStateModbusRead := - 1;
				
			//Error on Master, changes on Inputs or Timeout
		 	IF timTimeout.Q THEN 
				iStateModbusError := 300; 
					 
			END_IF
	
END_CASE

(*------------------------------------------------------------------Error and Warning----------------------------------------------------------------------------*)	
 
IF wStationState = 10 OR arrConnectorState[1] = 10 OR arrConnectorState[2] = 10 OR arrConnectorState[3] = 10 OR arrConnectorState[4] = 10 THEN bErrorCS := TRUE; ELSE bErrorCS := FALSE; END_IF  

IF timDissableFunctions.Q THEN fbCS.bWarning := TRUE; fbCS.iWarningCode := 0; ELSE fbCS.bWarning := FALSE; END_IF   
	IF Lynus_Standards.GVL_Energy.stNumberOfDevices.diNumberOfECS > Constants_Energy.diMaxNumberOfElectricChargingStations OR bErrorCS OR bMBTCPError THEN 
		fbCS.bError := TRUE;
	ELSE 
		fbCS.bError := FALSE;
			fbCS.iErrorCode := 0;
	END_IF

IF Lynus_Standards.GVL_Energy.stNumberOfDevices.diNumberOfECS > Constants_Energy.diMaxNumberOfElectricChargingStations THEN fbCS.iErrorCode := 1;
ELSIF bErrorCS OR bMBTCPError THEN fbCS.iErrorCode := 0; END_IF

(*------------------------------------------------------------------Logic----------------------------------------------------------------------------*)

//Calcualte the total SOC if we have more then 1 battery in our system
diNumberOfActiveBatterys := 0;
	dwSumSOC := 0;
		FOR liLPBatteryData := 1 TO Constants_Energy.diMaxNumberOfBatterys BY 1 DO
			IF Lynus_Standards.GVL_Energy.stDataOfBatterys[diNrOfEMS_IN,liLPBatteryData].bEnabled THEN diNumberOfActiveBatterys := diNumberOfActiveBatterys + 1; END_IF
				dwSumSOC := dwSumSOC + Lynus_Standards.GVL_Energy.stDataOfBatterys[diNrOfEMS_IN,liLPBatteryData].dwSOC;
		END_FOR
	
IF diNumberOfActiveBatterys > 0 THEN
	fbCS.dwBatterySOC := DINT_TO_DWORD(DWORD_TO_DINT(dwSumSOC) / diNumberOfActiveBatterys);
ELSE
	fbCS.dwBatterySOC := 100;	//When we have no battery in the ems system
END_IF

//Check if one or more Batterysystems or batteryinverter make island mode
diNumberOfBatteryInverterInEPO := 0;
	FOR liLPInEPO := 1 TO Constants_Energy.diMaxNumberOfBatteryInverters BY 1 DO
		IF Lynus_Standards.GVL_Energy.stDataOfBatteryInverters[diNrOfEMS_IN,liLPInEPO].bWorkOnIslandMode THEN fbCS.bEPOIsActive := TRUE; diNumberOfBatteryInverterInEPO := diNumberOfBatteryInverterInEPO + 1; END_IF
	END_FOR 
		IF diNumberOfBatteryInverterInEPO <= 0 THEN fbCS.bEPOIsActive := FALSE; END_IF

//Digital input for external lock signal
fbDIExternalLock(bInvers:= FALSE, bSignal=> );

//Car connected to the ECS  
IF arrConnectorState[1] = 2 OR arrConnectorState[2] = 2 OR arrConnectorState[3] = 2 OR arrConnectorState[4] = 2 OR
	 arrConnectorState[1] = 3 OR arrConnectorState[2] = 3 OR arrConnectorState[3] = 3 OR arrConnectorState[4] = 3 OR 
		arrConnectorState[1] = 6 OR arrConnectorState[2] = 6 OR arrConnectorState[3] = 6 OR arrConnectorState[4] = 6 THEN 
		fbCS.bCarConnected := TRUE; 
ELSE 
		fbCS.bCarConnected := FALSE; 
END_IF 

//Charging time and SOC from the Car
fbCS.arrSocketChargingTimeInput[1] :=  arrChargingTime[1] / 60;
fbCS.arrSocketChargingTimeInput[2] :=  arrChargingTime[2] / 60;
fbCS.arrSocketChargingTimeInput[3] :=  arrChargingTime[3] / 60;
fbCS.arrSocketChargingTimeInput[4] :=  arrChargingTime[4] / 60;

fbCS.arrSOCCar[1] := arrSOCCar[1];
fbCS.arrSOCCar[2] := arrSOCCar[2];
fbCS.arrSOCCar[3] := arrSOCCar[3];
fbCS.arrSOCCar[4] := arrSOCCar[4];

//Mode 3 State
fbCS.arrSocketMode3StateECS[1] := '';
fbCS.arrSocketMode3StateECS[2] := '';
fbCS.arrSocketMode3StateECS[3] := '';
fbCS.arrSocketMode3StateECS[4] := '';
//ECS is Free
IF arrConnectorState[1] = 0 THEN fbCS.arrSocketMode3StateECS[1] := 'A'; END_IF
IF arrConnectorState[2] = 0 THEN fbCS.arrSocketMode3StateECS[2] := 'A'; END_IF
IF arrConnectorState[3] = 0 THEN fbCS.arrSocketMode3StateECS[3] := 'A'; END_IF
IF arrConnectorState[4] = 0 THEN fbCS.arrSocketMode3StateECS[4] := 'A'; END_IF
//ECS Car Connected
IF arrConnectorState[1] = 2 OR arrConnectorState[1] = 6 THEN fbCS.arrSocketMode3StateECS[1] := 'B1'; END_IF
IF arrConnectorState[2] = 2 OR arrConnectorState[2] = 6 THEN fbCS.arrSocketMode3StateECS[2] := 'B1'; END_IF
IF arrConnectorState[3] = 2 OR arrConnectorState[3] = 6 THEN fbCS.arrSocketMode3StateECS[3] := 'B1'; END_IF
IF arrConnectorState[4] = 2 OR arrConnectorState[4] = 6 THEN fbCS.arrSocketMode3StateECS[4] := 'B1'; END_IF
//ECS Car is Charging
IF arrConnectorState[1] = 3 THEN fbCS.arrSocketMode3StateECS[1] := 'C2'; END_IF
IF arrConnectorState[2] = 3 THEN fbCS.arrSocketMode3StateECS[2] := 'C2'; END_IF
IF arrConnectorState[3] = 3 THEN fbCS.arrSocketMode3StateECS[3] := 'C2'; END_IF
IF arrConnectorState[4] = 3 THEN fbCS.arrSocketMode3StateECS[4] := 'C2'; END_IF

//Functionblock ECS
fbCS(
	bEnable:= bEnable AND NOT timDissableFunctions.Q, 
	bError:= ,
	bWarning := ,
	bEPOIsActive:= , 
	bExternalLock:= fbDIExternalLock.bSignal, 
	bCarConnected:= , 
	bWriteWithDelay:= TRUE, 
	bCalculateEnergySession:= ,
	iErrorCode:= , 
	iWarningCode:= , 
	arrSocketChargingTimeInput:= ,
	arrSOCCar:= , 
	dwBatterySOC:= , 
	lrTotalCounterEnergy_Consumption:= , 
	lrTotalCounterEnergy_Production:= , 
	lrCounterEnergyT1_Consumption:= , 
	lrCounterEnergyT2_Consumption:= , 
	lrCounterEnergyT1_Production:= , 
	lrCounterEnergyT2_Production:= , 
	lrTotalPowerECS:= , 
	arrSocketEnergySession:= ,
	rTargetPower:= Lynus_Standards.GVL_Energy.stDataElectricChargingStations[diNrOfEMS_IN,diNrOfECS_OUT].rTargetPowerEMS, 
	rSupplyVoltage:= 692, 
	rMinCurrent:= 7.5, 
	tTimDelayOutput:= T#5S, 
	tDelayError:= T#5S,
	arrSocketMode3StateECS:= ,
	arrSocketPowerECS:= ,
	stSetupECS:= stSetupECS, 
	stDataECSOut=> , 
	stDataECSOutDelay=> stDataECS);

dwTargetPower := REAL_TO_DWORD((stSetupECS.rMaxPower * fbCS.stDataECSOut.rTargetPower) / 100);
	dwTargetPower := dwTargetPower * 1000;

//Real time Power for Output
lrTotalPowerECSRealTime := fbCS.stDataECSOut.lrTotalPower;
	
(*------------------------------------------------------------------------------------------State Machine Write---------------------------------------------------------------------------------------------*)	

CASE iStateModbusWrite OF	

	1://Set the charging power (Reg 0)
		iStateModbus_CP := iStateModbusWrite;
		
			fbMBWrite_FC16.nQuantity := 2;
				fbMBWrite_FC16.nMBAddr := 0;
					fbMBWrite_FC16.bExecute := TRUE;
						fbMBWrite_FC16.nUnitID := byUnitID;
		
		//Prepear the sending Data. Charging Power for the charging station. 
		//Charging power
		fbConvertDwordToWord(dwInputValue:= dwTargetPower, eByteOrderForConvert:= eByteOrder.eBigEndian, wOutputValue_1=> arrBuffer_FC16[1], wOutputValue_2=> arrBuffer_FC16[2]);
		
		IF fbMBWrite_FC16.bBusy THEN timDelay.IN := TRUE; END_IF

		//Wait for Delay and then next step
		IF NOT fbMBWrite_FC16.bBusy AND NOT fbMBWrite_FC16.bError AND timDelay.Q THEN
			fbMBWrite_FC16.bExecute := FALSE;
				timDelay.IN := FALSE;
					bMBTCPError := FALSE; 
						//Restart from new with the Read out part
						iStateModbusRead := 1;
							iStateModbusWrite := 0;
								wConnectorInProgress := wConnectorInProgress + 1;
									IF wConnectorInProgress > 4 OR wConnectorInProgress > wNumberOfConnectors THEN wConnectorInProgress := 1; END_IF
		END_IF
				
		//Error or Timout
		IF FPError_FC_16.Q OR timTimeout.Q THEN
			iStateModbusError := 300;
		END_IF
		
END_CASE	
	
(*------------------------------------------------------------------------------------------State Machine Error---------------------------------------------------------------------------------------------*)	

CASE iStateModbusError OF
	
	300://Error
		iStateModbus_CP := iStateModbusError;
			timDelay.IN := FALSE;
				fbMBRead_FC4.bExecute := FALSE;
					fbMBWrite_FC16.bExecute := FALSE;
						bMBTCPError := TRUE; 		
							//Restart from new with the Read out part after an Error
							iStateModbusRead := 1;	
								iStateModbusError := 0;
									iStateModbusWrite := 0;
						
END_CASE

(*------------------------------------------------------------------------------------------Modbus TCP Functions---------------------------------------------------------------------------------------------*)

fbMBRead_FC4(sIPAddr:= sIPAdress, nTCPPort:= 502,cbLength:= SIZEOF(arrBuffer_FC4), pDestAddr:= ADR(arrBuffer_FC4), tTimeout:= T#10S );
	FPError_FC_4(CLK:= fbMBRead_FC4.bError, Q=> );		

fbMBWrite_FC16(sIPAddr:= sIPAdress, nTCPPort:= 502, cbLength:= SIZEOF(arrBuffer_FC16), pSrcAddr:= ADR(arrBuffer_FC16), tTimeout:= T#10S);	
	FPError_FC_16(CLK:= fbMBWrite_FC16.bError, Q=> );

(*-----------------------------------------------------------Handle data to Global structure for electric charging stations-----------------------------------------------------------------*)

//Delte al old Data on GVL after a online change or change on the variable diNrOfEMS_IDOD
IF diNrOfEMS_IN <> diNrOfEMS_IN_CP AND iStateGVLData = 0 THEN iStateGVLData := 10; END_IF 

CASE iStateGVLData OF
	
	0://Init Step
		byWaitInStep := 0;
			diCounterForGVL := 1;
	
	1://Wait for 4 Steps before clean al Data on GVL
		byWaitInStep := byWaitInStep + 1;
			IF byWaitInStep >= 4 AND fbNumberDevice.bNumberIsCalculatet THEN iStateGVLData := 2; END_IF
				//To much Devices, back to the Init step
				IF byWaitInStep >= 4 AND NOT fbNumberDevice.bNumberIsCalculatet THEN iStateGVLData := 0; END_IF	
			
	2://Clear all Data in GVL
		FOR diLPForGVL := 1 TO Constants_Energy.diMaxNumberOfEMS BY 1 DO 
			Lynus_Standards.GVL_Energy.stDataElectricChargingStations[diLPForGVL,diCounterForGVL].bEnabled := FALSE;
				Lynus_Standards.GVL_Energy.stDataElectricChargingStations[diLPForGVL,diCounterForGVL].bIsControllable := FALSE;
					Lynus_Standards.GVL_Energy.stDataElectricChargingStations[diLPForGVL,diCounterForGVL].byErrorWarning := 0;
						Lynus_Standards.GVL_Energy.stDataElectricChargingStations[diLPForGVL,diCounterForGVL].byPriority := 0;
							Lynus_Standards.GVL_Energy.stDataElectricChargingStations[diLPForGVL,diCounterForGVL].lrPower := 0;
								Lynus_Standards.GVL_Energy.stDataElectricChargingStations[diLPForGVL,diCounterForGVL].lrPowerConsumption := 0;
									Lynus_Standards.GVL_Energy.stDataElectricChargingStations[diLPForGVL,diCounterForGVL].lrPowerProduction := 0;
										Lynus_Standards.GVL_Energy.stDataElectricChargingStations[diLPForGVL,diCounterForGVL].rMaxPower := 0;
											//Set also the target value from ems back here to 0 and not in EMS function because EMS is in Standy when we have a online change (Problem when we delete a ems function and make a online change)
											Lynus_Standards.GVL_Energy.stDataElectricChargingStations[diLPForGVL,diCounterForGVL].rTargetPowerEMS := 0;	
		END_FOR
		
			//Counter for ECS
			diCounterForGVL := diCounterForGVL + 1;
				diCounterForGVL := LIMIT(0,diCounterForGVL,Constants_Energy.diMaxNumberOfElectricChargingStations);
					//Back to the init step
					IF diCounterForGVL >= Constants_Energy.diMaxNumberOfElectricChargingStations THEN iStateGVLData := 0; END_IF

	10://Clear old Data on GVL 		
		Lynus_Standards.GVL_Energy.stDataElectricChargingStations[diNrOfEMS_IN_CP,diNrOfECS_OUT].bEnabled := FALSE;
			Lynus_Standards.GVL_Energy.stDataElectricChargingStations[diNrOfEMS_IN_CP,diNrOfECS_OUT].bIsControllable := FALSE;
				Lynus_Standards.GVL_Energy.stDataElectricChargingStations[diNrOfEMS_IN_CP,diNrOfECS_OUT].byErrorWarning := 0;
					Lynus_Standards.GVL_Energy.stDataElectricChargingStations[diNrOfEMS_IN_CP,diNrOfECS_OUT].byPriority := 0;
						Lynus_Standards.GVL_Energy.stDataElectricChargingStations[diNrOfEMS_IN_CP,diNrOfECS_OUT].lrPower := 0;
							Lynus_Standards.GVL_Energy.stDataElectricChargingStations[diNrOfEMS_IN_CP,diNrOfECS_OUT].lrPowerConsumption := 0;
								Lynus_Standards.GVL_Energy.stDataElectricChargingStations[diNrOfEMS_IN_CP,diNrOfECS_OUT].lrPowerProduction := 0;
									Lynus_Standards.GVL_Energy.stDataElectricChargingStations[diNrOfEMS_IN_CP,diNrOfECS_OUT].rMaxPower := 0;
									
		diNrOfEMS_IN_CP := diNrOfEMS_IN;
			//Back to the init step
			iStateGVLData := 0;

END_CASE 	 

IF diNrOfECS_OUT > 0 AND fbNumberDevice.bNumberIsCalculatet AND diNrOfEMS_IN > 0 THEN
	Lynus_Standards.GVL_Energy.stDataElectricChargingStations[diNrOfEMS_IN,diNrOfECS_OUT].bEnabled := fbCS.stDataECSOut.bEnabled;
		Lynus_Standards.GVL_Energy.stDataElectricChargingStations[diNrOfEMS_IN,diNrOfECS_OUT].bIsControllable := TRUE;
			Lynus_Standards.GVL_Energy.stDataElectricChargingStations[diNrOfEMS_IN,diNrOfECS_OUT].byErrorWarning := fbCS.stDataECSOut.byErrorWarning;
				Lynus_Standards.GVL_Energy.stDataElectricChargingStations[diNrOfEMS_IN,diNrOfECS_OUT].byPriority := fbCS.stDataECSOut.byPriority;
					Lynus_Standards.GVL_Energy.stDataElectricChargingStations[diNrOfEMS_IN,diNrOfECS_OUT].lrPower := fbCS.stDataECSOut.lrTotalPower;
						Lynus_Standards.GVL_Energy.stDataElectricChargingStations[diNrOfEMS_IN,diNrOfECS_OUT].lrPowerConsumption := fbCS.stDataECSOut.lrTotalPowerConsumption;
							Lynus_Standards.GVL_Energy.stDataElectricChargingStations[diNrOfEMS_IN,diNrOfECS_OUT].lrPowerProduction := fbCS.stDataECSOut.lrTotalPowerProduction;
								Lynus_Standards.GVL_Energy.stDataElectricChargingStations[diNrOfEMS_IN,diNrOfECS_OUT].rMaxPower := fbCS.stDataECSOut.rMaxPower;	
END_IF 

(*----------------------------------------------------------Save persistent data----------------------------------------------------------------*)

arrPD[1](lrValue:= BOOL_TO_LREAL(bEnable), bEventBasedActive=> );
arrPD[2](lrValue:= BOOL_TO_LREAL(bPowerDataInvers), bEventBasedActive=> );
arrPD[3](lrValue:= DINT_TO_LREAL(diNrOfEMS_IN), bEventBasedActive=> );
arrPD[4](lrValue:= DINT_TO_LREAL(diNrOfEM_IN_CS), bEventBasedActive=> );
arrPD[5](lrValue:= BOOL_TO_LREAL(stSetupECS.bManualyOn), bEventBasedActive=> );
arrPD[6](lrValue:= BOOL_TO_LREAL(stSetupECS.bOnEmergPowerOff), bEventBasedActive=> );
arrPD[7](lrValue:= BYTE_TO_LREAL(stSetupECS.byCSMinPower), bEventBasedActive=> );
arrPD[8](lrValue:= BYTE_TO_LREAL(stSetupECS.byDisableSOC), bEventBasedActive=> );
arrPD[9](lrValue:= BYTE_TO_LREAL(stSetupECS.byEnableSOC), bEventBasedActive=> );
arrPD[10](lrValue:= BYTE_TO_LREAL(stSetupECS.byManualyTargetPower), bEventBasedActive=> );
arrPD[11](lrValue:= BYTE_TO_LREAL(stSetupECS.byPriority), bEventBasedActive=> );
arrPD[12](lrValue:= REAL_TO_LREAL(stSetupECS.rMaxPower), bEventBasedActive=> );
arrPD[13](lrValue:= DINT_TO_LREAL(diNrOfEMS_IN_CP), bEventBasedActive=> );
arrPD[14](lrValue:= BYTE_TO_LREAL(byUnitID), bEventBasedActive=> );
fbPDString(sText:= sIPAdress, bEventBasedActive=> );

END_FUNCTION_BLOCK

// ---- FB/FB_ElectricChargingStation_1.TcPOU

FUNCTION_BLOCK FB_ElectricChargingStation_1
VAR_INPUT
	
	bEnable									: BOOL;									//Enable the Fuctionblock and his logic
	
	bError									: BOOL;									//Error Input charging station
	
	bWarning								: BOOL;									//Warning Input charging station
	
	bEPOIsActive							: BOOL;									//Emergency power operation is active
	
	bExternalLock							: BOOL;									//External lock (All functions are locked)
	
	bCarConnected							: BOOL;									//Feedback if the car is connected to the charging station
	
	bWriteWithDelay							: BOOL;									//Write with Delay the Data to the output (Not al Output Data is writen with Delay)
	
	bCalculateEnergySession					: BOOL;									//When its true then the Energy Session is calculatet by the diffference of arrEnergySession[] when we have a change. FALSE = Use direct the Input from arrEnergySession[]
	
	iErrorCode								: INT;									//Error Code from external ECS
	
	iWarningCode							: INT;									//Warning Code from external ECS
								
	dwBatterySOC							: DWORD;								//Actual Battery SOC in %
	
	lrTotalCounterEnergy_Consumption		: LREAL;								//Total Counter for Energy consumption with unit Wh
	
	lrTotalCounterEnergy_Production			: LREAL;								//Total Counter for Energy production with unit Wh
	
	lrCounterEnergyT1_Consumption			: LREAL;								//Total counter for energy Tariff 1 consumption with unit Wh
	
	lrCounterEnergyT2_Consumption			: LREAL;								//Total counter for energy Tariff 2 consumption with unit Wh
	
	lrCounterEnergyT1_Production			: LREAL;								//Total counter for energy Tariff 1 production with unit Wh
	
	lrCounterEnergyT2_Production			: LREAL;								//Total counter for energy Tariff 2 production with unit Wh
	
	lrTotalPowerECS							: LREAL;								//Input Value from the total power of the charging station with unit W
	
	rTargetPower							: REAL;									//Target power from 0% to +100%
	
	rSupplyVoltage							: REAL;									//Supply voltage of the charging station for current calculation
	
	rMinCurrent								: REAL;									//Min. current that must flow for the charging station to switch on (if the current falls below this value, the car will not accept charging)
	
	tTimDelayOutput							: TIME := T#5S;							//Delay Time to write some Data to the Output	
	
	tDelayError								: TIME := T#15S;						//Delay for Error
		
	arrSocketMode3StateECS					: ARRAY[1..4] OF STRING(2);				//Mode 3 State Charging Station of each socket (A + E = ECS Ready or free, B1 + B2 + C1 + D1 = Car connected, C2 + D2 = Charging, F = Error)
		
	arrSOCCar								: ARRAY[1..4] OF DWORD;					//SOC from the car from each socket. 0 - 100%
		
	arrSocketChargingTimeInput				: ARRAY[1..4] OF REAL;					//Past charging time in min from each socket
		
	arrSocketEnergySession					: ARRAY[1..4] OF LREAL;					//Input for Energy Session or total Energy Counter of each socket. Look at the Input bCalculateEnergySession. Wh
		
	arrSocketPowerECS						: ARRAY[1..4] OF LREAL;					//Input Value from the power of each socket from the charging station with unit W
	
	stSetupECS								: ST_Setup_ECS;							//Setup charging station
END_VAR
VAR_OUTPUT
	
	stDataECSOut							: ST_ECS_Output;						//Electric charging station output data
	
	stDataECSOutDelay						: ST_ECS_Output;						//Electric charging station output data with delay
END_VAR
VAR
	FPEnable								: R_TRIG;								//Internal positive Edge
	FNManualy								: F_TRIG;								//Internal negative edge
	FNEnable								: F_TRIG;								//Internal negative Edge
	timDelayOutputs							: TON;									//Timer to send Data with Delay to the outputs
	timError								: TON;									//Timer to set the error
	timSOCDissable							: TON;									//Delay to dissable the ECS when the battery SOC has reached the value to dissale
	bMinCurrent								: BOOL;									//Current is fallen below min
	rMaxCurrent								: REAL;									//Max current from the charging station
	rPorcentOn								: REAL;									//Porcent value when the charging station switch on
	FPMode3C2								: ARRAY[1..4] OF R_TRIG;				//Internal positive Edge
	FPMode3D2								: ARRAY[1..4] OF R_TRIG;				//Internal positive Edge
	arrEnergySession_Cmp					: ARRAY[1..4] OF LREAL;					//Total Energy Comsumption for calculation of the energy session
END_VAR

//Creator : Kai Ebensperger
//Company : Lynus AG
//Date : 19.05.2021
//Version : 1.0.0.0

//This function block can be used to display the basic logic of a charging station.
//The charging station can either be switched on manually, in which case the power specification is not observed
//Otherwise the switching output of the charging station is set at 100% power setting
//In the power default mode, the SOC of the battery must be between On and Off SOC and must have reached On SOC once
//< Constants.byTargetOffPowerOnOffDevices the output is reset because of the hysteresis
//This FB can be used for charging stations on/off and for those which can be controlled linearly.
//Furthermore, the FB has an external blocking signal which switches off all functions as long as this is active.
//In addition, the FB outputs the power specification in parallel as a current specification. Ratio between power and voltage

(*---------------------------------------------------------------Check the limits of the inputs-------------------------------------------------------------------------------*)

arrSOCCar[1] := LIMIT(0,arrSOCCar[1],100); arrSOCCar[2] := LIMIT(0,arrSOCCar[2],100); arrSOCCar[3] := LIMIT(0,arrSOCCar[3],100); arrSOCCar[4] := LIMIT(0,arrSOCCar[4],100);
	dwBatterySOC := LIMIT(0,dwBatterySOC,100);
		rTargetPower := LIMIT(0,rTargetPower,100);
			stSetupECS.byManualyTargetPower := LIMIT(0,stSetupECS.byManualyTargetPower,100);
				stSetupECS.rMaxPower := LIMIT(0,stSetupECS.rMaxPower,500);
					stSetupECS.byCSMinPower := LIMIT(0,stSetupECS.byCSMinPower,100);	
						arrSocketChargingTimeInput[1] := LIMIT(0,arrSocketChargingTimeInput[1],100000); arrSocketChargingTimeInput[2] := LIMIT(0,arrSocketChargingTimeInput[2],100000); arrSocketChargingTimeInput[3] := LIMIT(0,arrSocketChargingTimeInput[3],100000); arrSocketChargingTimeInput[4] := LIMIT(0,arrSocketChargingTimeInput[4],100000);
							rSupplyVoltage := LIMIT(0,rSupplyVoltage,1000);
							
IF IsFinite(F_LREAL(lrTotalCounterEnergy_Consumption)) THEN lrTotalCounterEnergy_Consumption := LIMIT(0,lrTotalCounterEnergy_Consumption,999999999999999); END_IF
	IF IsFinite(F_LREAL(lrTotalCounterEnergy_Production)) THEN lrTotalCounterEnergy_Production := LIMIT(0,lrTotalCounterEnergy_Production,999999999999999); END_IF
		IF IsFinite(F_LREAL(lrCounterEnergyT1_Consumption)) THEN lrCounterEnergyT1_Consumption := LIMIT(0,lrCounterEnergyT1_Consumption,999999999999999); END_IF
			IF IsFinite(F_LREAL(lrCounterEnergyT2_Consumption)) THEN lrCounterEnergyT2_Consumption := LIMIT(0,lrCounterEnergyT2_Consumption,999999999999999); END_IF
				IF IsFinite(F_LREAL(lrCounterEnergyT1_Production)) THEN lrCounterEnergyT1_Production := LIMIT(0,lrCounterEnergyT1_Production,999999999999999); END_IF
					IF IsFinite(F_LREAL(lrCounterEnergyT2_Production)) THEN lrCounterEnergyT2_Production := LIMIT(0,lrCounterEnergyT2_Production,999999999999999); END_IF
						lrTotalPowerECS := LIMIT(-999999999999999,lrTotalPowerECS,999999999999999);
							arrSocketPowerECS[1] := LIMIT(-999999999999999,arrSocketPowerECS[1],999999999999999);
								arrSocketPowerECS[2] := LIMIT(-999999999999999,arrSocketPowerECS[2],999999999999999);
									arrSocketPowerECS[3] := LIMIT(-999999999999999,arrSocketPowerECS[3],999999999999999);
										arrSocketPowerECS[4] := LIMIT(-999999999999999,arrSocketPowerECS[4],999999999999999);
											IF IsFinite(F_LREAL(arrSocketEnergySession[1])) THEN arrSocketEnergySession[1] := LIMIT(0,arrSocketEnergySession[1],999999999999999); END_IF
												IF IsFinite(F_LREAL(arrSocketEnergySession[2])) THEN arrSocketEnergySession[2] := LIMIT(0,arrSocketEnergySession[2],999999999999999); END_IF
													IF IsFinite(F_LREAL(arrSocketEnergySession[3])) THEN arrSocketEnergySession[3] := LIMIT(0,arrSocketEnergySession[3],999999999999999); END_IF
														IF IsFinite(F_LREAL(arrSocketEnergySession[4])) THEN arrSocketEnergySession[4] := LIMIT(0,arrSocketEnergySession[4],999999999999999); END_IF
					
IF stSetupECS.byDisableSOC > stSetupECS.byEnableSOC THEN stSetupECS.byEnableSOC := stSetupECS.byDisableSOC + 1; END_IF

stSetupECS.byDisableSOC := LIMIT(0,stSetupECS.byDisableSOC,100);
	stSetupECS.byEnableSOC := LIMIT(1,stSetupECS.byEnableSOC,100);

(*---------------------------------------------------------------------------Enable----------------------------------------------------------------------------------*)

stDataECSOut.bEnabled := bEnable;

(*-----------------------------------------------------------------------------Error and Warning----------------------------------------------------------------------------*)

timError(IN:= bError, PT:= tDelayError, Q=> , ET=> );

stDataECSOut.byErrorWarning := 0;
	IF bWarning THEN stDataECSOut.byErrorWarning := 1; END_IF 
	IF timError.Q THEN stDataECSOut.byErrorWarning := 2; END_IF

//Messages and Error Codes
IF bExternalLock THEN stDataECSOut.eMessage := E_Message_ECS.eExternalLockActive;
ELSIF stDataECSOut.byErrorWarning = 1 AND iWarningCode = 0 THEN stDataECSOut.eMessage := E_Message_ECS.eNoConnectionToBackend;
ELSIF stDataECSOut.byErrorWarning = 1 AND iWarningCode = 1 THEN stDataECSOut.eMessage := E_Message_ECS.eWarningECS;
ELSIF stDataECSOut.byErrorWarning = 2 AND iErrorCode = 0 THEN stDataECSOut.eMessage := E_Message_ECS.eErrorECS;
ELSIF stDataECSOut.byErrorWarning = 2 AND iErrorCode = 1 THEN stDataECSOut.eMessage := E_Message_ECS.eTooMuchECS;
ELSE stDataECSOut.eMessage := E_Message_ECS.eNoMessage; 
END_IF

(*----------------------------------------------------------------------------Logic Part------------------------------------------------------------------------------------*)

//Target power
stDataECSOut.rTargetPower := DINT_TO_REAL(REAL_TO_DINT(rTargetPower * 100)) / 100;
IF rTargetPower <= stSetupECS.byCSMinPower THEN stDataECSOut.rTargetPower := BYTE_TO_REAL(stSetupECS.byCSMinPower); END_IF 
IF stSetupECS.bManualyOn THEN stDataECSOut.rTargetPower := BYTE_TO_REAL(stSetupECS.byManualyTargetPower); END_IF  

//When the current is fallen below the minimum then the charging station is switching off
//Calculate the max current for this charging station
IF rSupplyVoltage > 0 THEN
	rMaxCurrent := (stSetupECS.rMaxPower * 1000) / rSupplyVoltage;
ELSE
	rMaxCurrent := 0;
END_IF
	stDataECSOut.rTargetChargeCurrent := F_Scalvalue(x:= stDataECSOut.rTargetPower, x1:= 0, y1:= 0, x2:= 100, y2:= rMaxCurrent); 
	
IF rMaxCurrent = 0 THEN bMinCurrent := TRUE; ELSE bMinCurrent := FALSE; END_IF

//Calculate the porcent value for the min current
IF rMaxCurrent > 0 THEN
	rPorcentOn := (100 * rMinCurrent) / rMaxCurrent;
ELSE
	rPorcentOn := 0;
END_IF

//Timer for SOC Dissable
timSOCDissable(IN:= dwBatterySOC <= stSetupECS.byDisableSOC, PT:= T#30S, Q=> , ET=> );
	
//Switch Off
FNManualy(CLK:= stSetupECS.bManualyOn, Q=> ); 

IF NOT bEnable OR bMinCurrent OR bExternalLock OR stDataECSOut.byErrorWarning = 2 OR stDataECSOut.rTargetPower <= 0 OR timSOCDissable.Q OR (bEPOIsActive AND stSetupECS.bOnEmergPowerOff) OR FNManualy.Q THEN
	stDataECSOut.bOutput := FALSE;
END_IF

//Switch On
IF (bEnable AND NOT bExternalLock AND stDataECSOut.byErrorWarning <> 2 AND NOT bMinCurrent AND NOT bEPOIsActive AND stDataECSOut.rTargetPower > rPorcentOn AND dwBatterySOC >= stSetupECS.byEnableSOC) OR 
	(bEnable AND NOT bExternalLock AND stDataECSOut.byErrorWarning <> 2 AND bEPOIsActive AND NOT bMinCurrent AND NOT stSetupECS.bOnEmergPowerOff AND stDataECSOut.rTargetPower > rPorcentOn AND dwBatterySOC >= stSetupECS.byEnableSOC) OR
		(bEnable AND NOT bExternalLock AND NOT bMinCurrent AND stDataECSOut.byErrorWarning <> 2 AND stSetupECS.bManualyOn AND stDataECSOut.rTargetPower > rPorcentOn) THEN	
			stDataECSOut.bOutput := TRUE;
END_IF 

//Use this Output to switch Charging station on and off without possibility to send a target power value (Not controllable)
IF stDataECSOut.rTargetPower >= 100 AND stDataECSOut.bOutput THEN stDataECSOut.bOutputOnOff := TRUE; END_IF  
IF stDataECSOut.rTargetPower < Constants_Energy.byTargetOffPowerForOnOffDevices OR NOT stDataECSOut.bOutput THEN stDataECSOut.bOutputOnOff := FALSE; END_IF  

IF NOT stDataECSOut.bOutput THEN stDataECSOut.rTargetPower := 0; stDataECSOut.rTargetChargeCurrent := 0; END_IF 

IF stDataECSOut.rTargetChargeCurrent < rMinCurrent AND stDataECSOut.bOutput THEN stDataECSOut.rTargetChargeCurrent := rMinCurrent; END_IF

stDataECSOut.rTargetChargeCurrent := DINT_TO_REAL(REAL_TO_DINT(stDataECSOut.rTargetChargeCurrent * 100)) / 100;

(*------------------------------------------------------------------Power data----------------------------------------------------------------------------------------------*)

IF bEnable THEN
	stDataECSOut.lrTotalPower:= LINT_TO_LREAL(LREAL_TO_LINT((lrTotalPowerECS / 1000) * 100)) / 100;
		IF IsFinite(F_LREAL(lrCounterEnergyT1_Consumption)) THEN stDataECSOut.lrCounterEnergyT1_Consumption := LINT_TO_LREAL(LREAL_TO_LINT((lrCounterEnergyT1_Consumption / 1000) * 100)) / 100; END_IF
			IF IsFinite(F_LREAL(lrCounterEnergyT2_Consumption)) THEN stDataECSOut.lrCounterEnergyT2_Consumption := LINT_TO_LREAL(LREAL_TO_LINT((lrCounterEnergyT2_Consumption / 1000) * 100)) / 100; END_IF
				IF IsFinite(F_LREAL(lrCounterEnergyT1_Production)) THEN stDataECSOut.lrCounterEnergyT1_Production := LINT_TO_LREAL(LREAL_TO_LINT((lrCounterEnergyT1_Production / 1000) * 100)) / 100; END_IF
					IF IsFinite(F_LREAL(lrCounterEnergyT2_Production)) THEN stDataECSOut.lrCounterEnergyT2_Production := LINT_TO_LREAL(LREAL_TO_LINT((lrCounterEnergyT2_Production / 1000) * 100)) / 100; END_IF
						IF IsFinite(F_LREAL(lrTotalCounterEnergy_Consumption)) THEN stDataECSOut.lrTotalCounterEnergy_Consumption := LINT_TO_LREAL(LREAL_TO_LINT((lrTotalCounterEnergy_Consumption / 1000) * 100)) / 100; END_IF
							IF IsFinite(F_LREAL(lrTotalCounterEnergy_Production)) THEN stDataECSOut.lrTotalCounterEnergy_Production := LINT_TO_LREAL(LREAL_TO_LINT((lrTotalCounterEnergy_Production / 1000) * 100)) / 100; END_IF 
				
		IF stDataECSOut.lrTotalPower < 0 THEN
				stDataECSOut.lrTotalPowerProduction := (stDataECSOut.lrTotalPower * - 1);
				stDataECSOut.lrTotalPowerConsumption := 0;
		ELSIF stDataECSOut.lrTotalPower > 0 THEN
				stDataECSOut.lrTotalPowerProduction := 0;
				stDataECSOut.lrTotalPowerConsumption := stDataECSOut.lrTotalPower;
		ELSIF stDataECSOut.lrTotalPower = 0 THEN
				stDataECSOut.lrTotalPowerProduction := 0;
				stDataECSOut.lrTotalPowerConsumption := 0;
		END_IF
		
		//Socket Power
		stDataECSOut.arrSocketPower[1] := LINT_TO_LREAL(LREAL_TO_LINT((arrSocketPowerECS[1] / 1000) * 100)) / 100;
			stDataECSOut.arrSocketPower[2] := LINT_TO_LREAL(LREAL_TO_LINT((arrSocketPowerECS[2] / 1000) * 100)) / 100;
				stDataECSOut.arrSocketPower[3] := LINT_TO_LREAL(LREAL_TO_LINT((arrSocketPowerECS[3] / 1000) * 100)) / 100;
					stDataECSOut.arrSocketPower[4] := LINT_TO_LREAL(LREAL_TO_LINT((arrSocketPowerECS[4] / 1000) * 100)) / 100;
		
ELSE
	stDataECSOut.lrTotalPower := 0;
		stDataECSOut.lrCounterEnergyT1_Consumption := 0;
			stDataECSOut.lrCounterEnergyT2_Consumption := 0;
				stDataECSOut.lrCounterEnergyT1_Production := 0;
					stDataECSOut.lrCounterEnergyT2_Production := 0;
						stDataECSOut.lrTotalPowerProduction := 0;
							stDataECSOut.lrTotalPowerConsumption := 0;	
								stDataECSOut.lrTotalCounterEnergy_Consumption := 0;
									stDataECSOut.lrTotalCounterEnergy_Production := 0;
									
	//Socket
	stDataECSOut.arrSocketPower[1] := 0;
			stDataECSOut.arrSocketPower[2] := 0;
				stDataECSOut.arrSocketPower[3] := 0;
					stDataECSOut.arrSocketPower[4] := 0;
END_IF

//Calcualte Energy from actual Session
FPMode3C2[1](CLK:= arrSocketMode3StateECS[1] = 'C2', Q=> );
	FPMode3D2[1](CLK:= arrSocketMode3StateECS[1] = 'D2', Q=> );
		FPMode3C2[2](CLK:= arrSocketMode3StateECS[2] = 'C2', Q=> );
			FPMode3D2[2](CLK:= arrSocketMode3StateECS[2] = 'D2', Q=> );
				FPMode3C2[3](CLK:= arrSocketMode3StateECS[3] = 'C2', Q=> );
					FPMode3D2[3](CLK:= arrSocketMode3StateECS[3] = 'D2', Q=> );
						FPMode3C2[4](CLK:= arrSocketMode3StateECS[4] = 'C2', Q=> );
							FPMode3D2[4](CLK:= arrSocketMode3StateECS[4] = 'D2', Q=> );
			
IF bCalculateEnergySession THEN 
		//Socket 1
		IF FPMode3C2[1].Q OR FPMode3D2[1].Q THEN
			//Reset Counter when a new session is started
			stDataECSOut.arrSocketEnergySession[1] := 0;
				//Copy the Total Counter in kWh when a new session is started
				IF IsFinite(F_LREAL(arrSocketEnergySession[1])) THEN
					arrEnergySession_Cmp[1] := arrSocketEnergySession[1];
				END_IF
		END_IF
			IF (arrEnergySession_Cmp[1] <> arrSocketEnergySession[1] AND IsFinite(F_LREAL(arrSocketEnergySession[1])) AND (arrSocketMode3StateECS[1] = 'C2' OR arrSocketMode3StateECS[1] = 'D2')) THEN
				stDataECSOut.arrSocketEnergySession[1] := stDataECSOut.arrSocketEnergySession[1] + (arrSocketEnergySession[1] - arrEnergySession_Cmp[1]) / 1000;  
					stDataECSOut.arrSocketEnergySession[1] := stDataECSOut.arrSocketEnergySession[1];
						arrEnergySession_Cmp[1] := arrSocketEnergySession[1];		
			END_IF
		//Socket 2
		IF FPMode3C2[2].Q OR FPMode3D2[2].Q THEN
			//Reset Counter when a new session is started
			stDataECSOut.arrSocketEnergySession[2] := 0;
				//Copy the Total Counter in kWh when a new session is started
				IF IsFinite(F_LREAL(arrSocketEnergySession[2])) THEN
					arrEnergySession_Cmp[2] := arrSocketEnergySession[2];
				END_IF
		END_IF
			IF (arrEnergySession_Cmp[2] <> arrSocketEnergySession[2] AND IsFinite(F_LREAL(arrSocketEnergySession[2])) AND (arrSocketMode3StateECS[2] = 'C2' OR arrSocketMode3StateECS[2] = 'D2')) THEN
				stDataECSOut.arrSocketEnergySession[2] := stDataECSOut.arrSocketEnergySession[2] + (arrSocketEnergySession[2] - arrEnergySession_Cmp[2]) / 1000;  
					stDataECSOut.arrSocketEnergySession[2] := stDataECSOut.arrSocketEnergySession[2];
						arrEnergySession_Cmp[2] := arrSocketEnergySession[2];		
			END_IF
		//Socket 3
		IF FPMode3C2[3].Q OR FPMode3D2[3].Q THEN
			//Reset Counter when a new session is started
			stDataECSOut.arrSocketEnergySession[3] := 0;
				//Copy the Total Counter in kWh when a new session is started
				IF IsFinite(F_LREAL(arrSocketEnergySession[3])) THEN
					arrEnergySession_Cmp[3] := arrSocketEnergySession[3];
				END_IF
		END_IF
			IF (arrEnergySession_Cmp[3] <> arrSocketEnergySession[3] AND IsFinite(F_LREAL(arrSocketEnergySession[3])) AND (arrSocketMode3StateECS[3] = 'C2' OR arrSocketMode3StateECS[3] = 'D2')) THEN
				stDataECSOut.arrSocketEnergySession[3] := stDataECSOut.arrSocketEnergySession[3] + (arrSocketEnergySession[3] - arrEnergySession_Cmp[3]) / 1000;  
					stDataECSOut.arrSocketEnergySession[3] := stDataECSOut.arrSocketEnergySession[3];
						arrEnergySession_Cmp[3] := arrSocketEnergySession[3];		
			END_IF
		//Socket 4
		IF FPMode3C2[4].Q OR FPMode3D2[4].Q THEN
			//Reset Counter when a new session is started
			stDataECSOut.arrSocketEnergySession[4] := 0;
				//Copy the Total Counter in kWh when a new session is started
				IF IsFinite(F_LREAL(arrSocketEnergySession[4])) THEN
					arrEnergySession_Cmp[4] := arrSocketEnergySession[4];
				END_IF
		END_IF
			IF (arrEnergySession_Cmp[4] <> arrSocketEnergySession[4] AND IsFinite(F_LREAL(arrSocketEnergySession[4])) AND (arrSocketMode3StateECS[4] = 'C2' OR arrSocketMode3StateECS[4] = 'D2')) THEN
				stDataECSOut.arrSocketEnergySession[4] := stDataECSOut.arrSocketEnergySession[4] + (arrSocketEnergySession[4] - arrEnergySession_Cmp[4]) / 1000;  
					stDataECSOut.arrSocketEnergySession[4] := stDataECSOut.arrSocketEnergySession[4];
						arrEnergySession_Cmp[4] := arrSocketEnergySession[4];		
			END_IF
			
		stDataECSOut.arrSocketEnergySession[1] := LINT_TO_LREAL(LREAL_TO_LINT(stDataECSOut.arrSocketEnergySession[1] * 1000)) / 1000;
		stDataECSOut.arrSocketEnergySession[2] := LINT_TO_LREAL(LREAL_TO_LINT(stDataECSOut.arrSocketEnergySession[2] * 1000)) / 1000;
		stDataECSOut.arrSocketEnergySession[3] := LINT_TO_LREAL(LREAL_TO_LINT(stDataECSOut.arrSocketEnergySession[3] * 1000)) / 1000;
		stDataECSOut.arrSocketEnergySession[4] := LINT_TO_LREAL(LREAL_TO_LINT(stDataECSOut.arrSocketEnergySession[4] * 1000)) / 1000;
			
ELSE
	IF IsFinite(F_LREAL(arrSocketEnergySession[1])) THEN stDataECSOut.arrSocketEnergySession[1] := LINT_TO_LREAL(LREAL_TO_LINT((arrSocketEnergySession[1] / 1000) * 1000)) / 1000; END_IF
		IF IsFinite(F_LREAL(arrSocketEnergySession[2])) THEN stDataECSOut.arrSocketEnergySession[2] := LINT_TO_LREAL(LREAL_TO_LINT((arrSocketEnergySession[2] / 1000) * 1000)) / 1000; END_IF
			IF IsFinite(F_LREAL(arrSocketEnergySession[3])) THEN stDataECSOut.arrSocketEnergySession[3] := LINT_TO_LREAL(LREAL_TO_LINT((arrSocketEnergySession[3] / 1000) * 1000)) / 1000; END_IF
				IF IsFinite(F_LREAL(arrSocketEnergySession[4])) THEN stDataECSOut.arrSocketEnergySession[4] := LINT_TO_LREAL(LREAL_TO_LINT((arrSocketEnergySession[4] / 1000) * 1000)) / 1000; END_IF
END_IF
		
(*---------------------------------------------------------------------------Outputs--------------------------------------------------------------------------------------*)

stDataECSOut.byPriority := stSetupECS.byPriority;
	stDataECSOut.rMaxPower := DINT_TO_REAL(REAL_TO_DINT(stSetupECS.rMaxPower * 100)) / 100;
		stDataECSOut.bSOnEmergPowerOff := stSetupECS.bOnEmergPowerOff;
			stDataECSOut.bSManualyOn := stSetupECS.bManualyOn;
				stDataECSOut.bySManualyTargetPower := stSetupECS.byManualyTargetPower;
					stDataECSOut.bySCSMinPower := stSetupECS.byCSMinPower;

stDataECSOut.bCarConnected := bCarConnected;

//Mode 3 State
//Socket 1
//No Value.
IF arrSocketMode3StateECS[1] = '' OR arrSocketMode3StateECS[1] = 'F' OR NOT bEnable THEN
	stDataECSOut.arrSocketStateECS[1] := 0;
//ECS ready and Free	
ELSIF arrSocketMode3StateECS[1] = 'A' OR arrSocketMode3StateECS[1] = 'E' THEN
	stDataECSOut.arrSocketStateECS[1] := 1;
//Car Connected
ELSIF arrSocketMode3StateECS[1] = 'B1' OR arrSocketMode3StateECS[1] = 'B2' OR arrSocketMode3StateECS[1] = 'C1' OR arrSocketMode3StateECS[1] = 'D1' THEN
	stDataECSOut.arrSocketStateECS[1] := 2;
//Car Charging
ELSIF arrSocketMode3StateECS[1] = 'C2' OR arrSocketMode3StateECS[1] = 'D2' THEN
	stDataECSOut.arrSocketStateECS[1] := 3;
END_IF
//Socket 2
//No Value.
IF arrSocketMode3StateECS[2] = '' OR arrSocketMode3StateECS[2] = 'F' OR NOT bEnable THEN
	stDataECSOut.arrSocketStateECS[2] := 0;
//ECS ready and Free	
ELSIF arrSocketMode3StateECS[2] = 'A' OR arrSocketMode3StateECS[2] = 'E' THEN
	stDataECSOut.arrSocketStateECS[2] := 1;
//Car Connected
ELSIF arrSocketMode3StateECS[2] = 'B1' OR arrSocketMode3StateECS[2] = 'B2' OR arrSocketMode3StateECS[2] = 'C1' OR arrSocketMode3StateECS[2] = 'D1' THEN
	stDataECSOut.arrSocketStateECS[2] := 2;
//Car Charging
ELSIF arrSocketMode3StateECS[2] = 'C2' OR arrSocketMode3StateECS[2] = 'D2' THEN
	stDataECSOut.arrSocketStateECS[2] := 3;
END_IF
//Socket 3
//No Value.
IF arrSocketMode3StateECS[3] = '' OR arrSocketMode3StateECS[3] = 'F' OR NOT bEnable THEN
	stDataECSOut.arrSocketStateECS[3] := 0;
//ECS ready and Free	
ELSIF arrSocketMode3StateECS[3] = 'A' OR arrSocketMode3StateECS[3] = 'E' THEN
	stDataECSOut.arrSocketStateECS[3] := 1;
//Car Connected
ELSIF arrSocketMode3StateECS[3] = 'B1' OR arrSocketMode3StateECS[3] = 'B2' OR arrSocketMode3StateECS[3] = 'C1' OR arrSocketMode3StateECS[3] = 'D1' THEN
	stDataECSOut.arrSocketStateECS[3] := 2;
//Car Charging
ELSIF arrSocketMode3StateECS[3] = 'C2' OR arrSocketMode3StateECS[3] = 'D2' THEN
	stDataECSOut.arrSocketStateECS[3] := 3;
END_IF
//Socket 4
//No Value.
IF arrSocketMode3StateECS[4] = '' OR arrSocketMode3StateECS[4] = 'F' OR NOT bEnable THEN
	stDataECSOut.arrSocketStateECS[4] := 0;
//ECS ready and Free	
ELSIF arrSocketMode3StateECS[4] = 'A' OR arrSocketMode3StateECS[4] = 'E' THEN
	stDataECSOut.arrSocketStateECS[4] := 1;
//Car Connected
ELSIF arrSocketMode3StateECS[4] = 'B1' OR arrSocketMode3StateECS[4] = 'B2' OR arrSocketMode3StateECS[4] = 'C1' OR arrSocketMode3StateECS[4] = 'D1' THEN
	stDataECSOut.arrSocketStateECS[4] := 2;
//Car Charging
ELSIF arrSocketMode3StateECS[4] = 'C2' OR arrSocketMode3StateECS[4] = 'D2' THEN
	stDataECSOut.arrSocketStateECS[4] := 3;
END_IF
	
IF bEnable THEN
	stDataECSOut.arrSocketSOCCar[1] := arrSOCCar[1];
	stDataECSOut.arrSocketSOCCar[2] := arrSOCCar[2];
	stDataECSOut.arrSocketSOCCar[3] := arrSOCCar[3];
	stDataECSOut.arrSocketSOCCar[4] := arrSOCCar[4];
		stDataECSOut.arrChargingTimeInMin[1] := DINT_TO_REAL(REAL_TO_DINT(arrSocketChargingTimeInput[1] * 100)) / 100;
		stDataECSOut.arrChargingTimeInMin[2] := DINT_TO_REAL(REAL_TO_DINT(arrSocketChargingTimeInput[2] * 100)) / 100;
		stDataECSOut.arrChargingTimeInMin[3] := DINT_TO_REAL(REAL_TO_DINT(arrSocketChargingTimeInput[3] * 100)) / 100;
		stDataECSOut.arrChargingTimeInMin[4] := DINT_TO_REAL(REAL_TO_DINT(arrSocketChargingTimeInput[4] * 100)) / 100;
ELSE
	stDataECSOut.arrSocketSOCCar[1] := 0;
	stDataECSOut.arrSocketSOCCar[2] := 0;
	stDataECSOut.arrSocketSOCCar[3] := 0;
	stDataECSOut.arrSocketSOCCar[4] := 0;
		stDataECSOut.arrChargingTimeInMin[1] := 0;
		stDataECSOut.arrChargingTimeInMin[2] := 0;
		stDataECSOut.arrChargingTimeInMin[3] := 0;
		stDataECSOut.arrChargingTimeInMin[4] := 0;
END_IF

timDelayOutputs(IN:= bWriteWithDelay AND bEnable AND NOT timDelayOutputs.Q, PT:= tTimDelayOutput, Q=> , ET=> );
	FPEnable(CLK:= bEnable, Q=> );
		FNEnable(CLK:= bEnable, Q=> );
		
//Write with Delay or without
IF (bWriteWithDelay AND (timDelayOutputs.Q OR FPEnable.Q OR FNEnable.Q)) OR NOT bWriteWithDelay THEN
	stDataECSOutDelay := stDataECSOut;
END_IF

END_FUNCTION_BLOCK

// ---- POUs/prgPersistent.TcPOU
PROGRAM prgPersistent
VAR
	fbUSV		: FB_WritePersistentData_CX81xx;
	fb_Reboot		: NT_reboot;
	m_Reboot		: BOOL:=FALSE;
END_VAR

fbUSV(
	eSaveModeData:= eUSVSaveMode.eSaveWhenPowerfail, 
	bLoadPersistentDataOk=> , 
	bPowerFailDetect=> , 
	bError=> , 
	bySaveProcess=> , 
	dwStorageLast24h=> , 
	udiErrorCode=> );

	
fb_Reboot(	netid := '',
			delay := 2,
			start := m_Reboot);

END_PROGRAM

// ---- POUs/prgLynusCom.TcPOU
PROGRAM prgLynusCom
VAR
	fbCom		: FB_MqttCommunicator_V3;
	f_Trig_HB: f_trig;
	stringArray_Last_HB: ARRAY[0..50] OF STRING(30);
	intCount: INT;
	time_Temp: TIME;

END_VAR

fbCom(
	bConnect:= TRUE, 
	strAuthKey:=  'BMS99299754422' , 
	sUserName:= '34467fe1-3b9d-4cc2-8cff-1c321ed830b0', 
	sUserPassword:= '8cf1ce48-c398-49af-8d5b-32fb5d2a30fc', 
	eSavePositionCertificate:= eSavePositionOnPLC.ePostionHardDisk,
	time_HeartBeat_sec 		:= T#15S,
	bConnected=> , 
	bError=> , 
	hrErrorCode=> , 
	eConnectionState=> , 
	eErrorMessage_Out=> );
(*old
	sUserName:= '48e2db0e-41f9-4208-90bb-f2ed6b34cc1d', 
	sUserPassword:= 'd51f4679-bb87-4f59-a61e-f3f72e7e7746', 
*)
	
	
prg_SystemTime();
f_Trig_HB(CLK :=  fbCom.bHBSending);
IF f_Trig_HB.Q THEN
	IF intCount>50 OR intCount<0 THEN
		intCount:=0;
	END_IF
	stringArray_Last_HB[intCount] := prg_SystemTime.stringSystemTime_ms;
	intCount := intCount+1;
END_IF

time_Temp := fbCom.fbTimerHB.ET;

END_PROGRAM

// ---- FB/FB_Xelectrix_Powerbox_1.TcPOU
FUNCTION_BLOCK FB_Xelectrix_Powerbox_1
VAR_INPUT PERSISTENT
	bEnable							: BOOL;											//{#lynus.ag#()} //True = Function is enabled, FALSE = Function is dissabled, no new Data
	bActivateControl				: BOOL;											//Activate the control from the Xelectrix Inverter over Modbus TCP (False = Inverter work by himself)
	byUnitID						: BYTE;											//Unit ID fromt the Inverter (0 to 255)
	byPriority						: BYTE;											//{#lynus.ag#()} //Priority of the Device
	diNrOfEMS_IN					: DINT;											//Number of EMS what control this Device.
	lrMaxCapacityBattery			: LREAL;										//{#lynus.ag#()} //Max Capacity from the Battery in kWh. Here on this Function this Input Value cames from Inside of the Function.
	sIPAdress						: STRING(15);									//IP Adress from the Inverter
END_VAR
VAR_INPUT
	bReset							: BOOL;											//{#lynus.ag#()} //Reset the device after a Error or a Warning
END_VAR
VAR_OUTPUT
	stDataXelectrix					: ST_Xelectrix_Powerbox_OutData;				//Shows the specific output data from the Xelectric device
	stDataBatt						: ST_Battery_Output;							//{#lynus.ag#()} //Output structure with Data from Battery
	stDataBattInverter				: ST_BatteryInverter_Output;					//{#lynus.ag#()} //Output structure with Data from Battery Inverter
	stDataEMPower_Grid				: ST_ElectricMeter_Output_Power;				//Output structure with Data from Electric Meter Grid (Power Data)
	stDataEMCounter_Grid			: ST_ElectricMeter_Output_Counter;				//Output structure with Data from Electric Meter Grid (Counter Data)
	diNrOfBatt_OUT					: DINT;											//Active Number from the Battery Function for using on other functions
	diNrOfBattInverter_OUT			: DINT;											//Active Number from the Battery Inverter Function for using on other functions
	diNrOfEM_OUT_Grid				: DINT;											//Active Number from the Electric Meter for using on other functions
	lrMaxCapacityBattery_OUT		: LREAL;										//Max kWh from the Battery system. The Xelectrix System deliver this value.
END_VAR
VAR
	{attribute 'hide'}
	fbBattery						: FB_Battery;									//Function block for battery
	{attribute 'hide'}
	fbBatteryInverter				: FB_BatteryInverter;							//Function block for battery inveter
	{attribute 'hide'}
	fbEMGrid						: FB_ElectricMeter;								//Electric Meter Function 
	{attribute 'hide'}
	fbPIDChrgStandby				: FB_PID;										//Controller to control the battery current on 0 in the standby mode	
	{attribute 'hide'}
	fbNumberDeviceBattery			: FB_NumberOfDevice;							//Function block to calcualte the number of the Device
	{attribute 'hide'}
	fbNumberDeviceBatteryInvert		: FB_NumberOfDevice;							//Function block to calcualte the number of the Device
	{attribute 'hide'}
	fbNumberDeviceGrid				: FB_NumberOfDevice;							//Function block to calcualte the number of the Device
	{attribute 'hide'}
	fbMBRead_FC3					: FB_MBReadRegs;								//Modbus Read Function (FC3)
	{attribute 'hide'}
	fbMBWrite_FC16					: FB_MBWriteRegs;								//Modbus Write Function (FC16)
	{attribute 'hide'}
	fbConvertData					: FB_CV_WORD_TO_DWORD;							//Convert 2 Words in a Dword
	{attribute 'hide'}
	timDelay						: TON;											//Timer for Delay between Requests
	{attribute 'hide'}
	timTimeout						: TON;											//Timer for Timeout
	{attribute 'hide'}
	timDissableFunctions			: TON;											//Timer to dissable the Function after Lynus_Standards.Constants_General.tTimeDissableLynusFunctions Days without connection to the Lynus Cloud
	{attribute 'hide'}
	timResetConnectionOnGVL			: TON;											//Timer to try reset the connection Flag on the GVL. (When somebody delete the Connection Function and make only a onlinechange)
	{attribute 'hide'}
	timReset						: TON;											//Timer to reset the Inverter after a Error
	{attribute 'hide'}
	timErrorMTCP					: TON;											//Delay when Error on Modbus TCP
	{attribute 'hide'}
	timSetStandbyCntrl				: TOF;											//Timer to set the Standby Controller
	{attribute 'hide'}
	FPEnable						: R_TRIG;										//Internal positive Edge
	{attribute 'hide'}
	FPError_FC_3					: R_TRIG;										//Internal positive Edge
	{attribute 'hide'}
	FPError_FC_16					: R_TRIG;										//Internal positive Edge
	{attribute 'hide'}
	FPActivateControl				: R_TRIG;										//Internal positive Edge
	{attribute 'hide'}
	FNTimDissable					: F_TRIG;										//Internal negative Edge
	{attribute 'hide'}
	PD_String						: FB_PersistentData_String;						//Function to save persistent data
	{attribute 'hide'}
	arrPD							: ARRAY[1..7] OF FB_PersistentData_Number;		//Function to save persistent data
	{attribute 'hide'}
	arrBuffer_FC3					: ARRAY[1..48] OF WORD;							//Buffer with Data from FC3
	{attribute 'hide'}
	arrBuffer_FC16					: ARRAY[1..2] OF WORD;							//Buffer with Data from FC16
	{attribute 'hide'}
	arrCounterForGVL				: ARRAY[1..3] OF DINT;							//Counter to clean old data on GVL
	{attribute 'hide'}
	bEnergyGridConsReceived			: BOOL;											//Energy Consumption from Grid first time received
	{attribute 'hide'}
	bEnergyGridProdReceived			: BOOL;											//Energy Production from Grid first time received
	{attribute 'hide'}
	byWaitInStep					: BYTE;											//Wait in Step before start to clean data on PLC
	{attribute 'hide'}
	byLPWorkAroundACDevice			: BYTE;											//Loop for Workaround
	{attribute 'hide'}
	byNumberOfZero					: BYTE;											//Number with 0 Value from AC Messurement
	{attribute 'hide'}
	iSetpointPower					: INT;											//Power Setpoint in W
	{attribute 'hide'}
	iStateGVLData					: INT;											//State machine to handle the data on the GVL
	{attribute 'hide'}
	iStateModbusRead				: INT;											//State variable for Statemachine
	{attribute 'hide'}
	iStateModbusWrite				: INT;											//State variable for Statemachine
	{attribute 'hide'}
	iStateModbusError				: INT;											//State variable for Statemachine
	{attribute 'hide'}
	iStateModbus_CP					: INT;											//Compare State variable
	{attribute 'hide'}
	iMaxDcDischargeCurrentBattery	: INT;											//Variable to convert from negative to positive value
	{attribute 'hide'}
	diLPForGVL						: DINT;											//Loop to clean old data on GVL
	{attribute 'hide'}
	lrEnergyGridConsumption_CP		: LREAL;										//Energy Consumption from Grid for calculation for Workaround why Xelectrix send sometimes big value 
	{attribute 'hide'}
	lrEnergyGridProduction_CP		: LREAL;										//Energy Production from Grid for calculation for Workaround why Xelectrix send sometimes big value 
END_VAR
VAR PERSISTENT
	{attribute 'conditionalshow'}
	diNrOfEMS_IN_CP					: DINT;											//Number of EMS what control this Device to compare with the original
END_VAR

//Creator : Kai Ebensperger
//Company : Lynus AG
//Date : 30.06.2021
//Version : 1.0.0.0

//With this function its possible to read out values from the Xelectrix Powerbox from the factory Xelectrix
//Its also possible to controll the power in and out from Battery if its necessary.
//The protocol to the Inverter/powerbox is Modbus TCP
//When this Function is not enabled, then the Inverter is not off. But no power flows into or out of the battery.
//This Inverter deliver also the Grid power (smart Meter).
//Versions that are supported : 106
//NOTE : This Function block not support the complete emergency power mode. He switch not off when the byMaxDepthOfDischargeEPO is reached because this make the inverter by himself.

//NOTE for diNr.....Designation => 
//_IN = Here Data come in from other Functions or go out to other functions about the GVL
//_OUT = Here Data go out to other functions about the GVL

(*------------------------------------------------------------------------------------------General Input Part---------------------------------------------------------------------------------------------*)

//Check limitation
diNrOfEMS_IN := LIMIT(0,diNrOfEMS_IN,Constants_Energy.diMaxNumberOfEMS);
	
(*-------------------------------------------------------------Calcualte the number of Battery system---------------------------------------------------------------*)

fbNumberDeviceBattery(
	diActualNumberOfDevices:= Lynus_Standards.GVL_Energy.stNumberOfDevices.diNumberOfBatterys, 
	diMaxNumberOfDevices:= Constants_Energy.diMaxNumberOfBatterys, 
	udiCounterOnlineChange:= TwinCAT_SystemInfoVarList._AppInfo.OnlineChangeCnt, 
	bNumberIsCalculatet=> , 
	bFPNumberIsCalculatet=> , 
	bOnlineChange=> , 
	diNumberForThisDevice=> diNrOfBatt_OUT, 
	diNumberOfTotalDevices=> );

//Write new Numer on GVL
IF fbNumberDeviceBattery.bFPNumberIsCalculatet THEN
	Lynus_Standards.GVL_Energy.stNumberOfDevices.diNumberOfBatterys := fbNumberDeviceBattery.diNumberOfTotalDevices;	
END_IF

//Delete old Number on GVL
IF fbNumberDeviceBattery.bOnlineChange THEN 
	Lynus_Standards.GVL_Energy.stNumberOfDevices.diNumberOfBatterys := diNrOfBatt_OUT;	
		iStateGVLData := 1; 
END_IF

fbNumberDeviceBatteryInvert(
	diActualNumberOfDevices:= Lynus_Standards.GVL_Energy.stNumberOfDevices.diNumberOfBatteryInverters, 
	diMaxNumberOfDevices:= Constants_Energy.diMaxNumberOfBatteryInverters, 
	udiCounterOnlineChange:= TwinCAT_SystemInfoVarList._AppInfo.OnlineChangeCnt, 
	bNumberIsCalculatet=> , 
	bFPNumberIsCalculatet=> , 
	bOnlineChange=> , 
	diNumberForThisDevice=> diNrOfBattInverter_OUT, 
	diNumberOfTotalDevices=> );

//Write new Numer on GVL
IF fbNumberDeviceBatteryInvert.bFPNumberIsCalculatet THEN
	Lynus_Standards.GVL_Energy.stNumberOfDevices.diNumberOfBatteryInverters := fbNumberDeviceBatteryInvert.diNumberOfTotalDevices;	
END_IF

//Delete old Number on GVL
IF fbNumberDeviceBatteryInvert.bOnlineChange THEN 
	Lynus_Standards.GVL_Energy.stNumberOfDevices.diNumberOfBatteryInverters := diNrOfBattInverter_OUT;	
		iStateGVLData := 1; 
END_IF

fbNumberDeviceGrid(
	diActualNumberOfDevices:= Lynus_Standards.GVL_Energy.stNumberOfDevices.diNumberOfElectricMeters, 
	diMaxNumberOfDevices:= Constants_Energy.diMaxNumberOfElectricMeters, 
	udiCounterOnlineChange:= TwinCAT_SystemInfoVarList._AppInfo.OnlineChangeCnt, 
	bNumberIsCalculatet=> , 
	bFPNumberIsCalculatet=> , 
	bOnlineChange=> , 
	diNumberForThisDevice=> diNrOfEM_OUT_Grid, 
	diNumberOfTotalDevices=> );

//Write new Numer on GVL
IF fbNumberDeviceGrid.bFPNumberIsCalculatet THEN
	Lynus_Standards.GVL_Energy.stNumberOfDevices.diNumberOfElectricMeters := fbNumberDeviceGrid.diNumberOfTotalDevices;	
END_IF			

(*-------------------------------------------------------------Service from Backend is ready and check the connection to backend for dissabel/enable Function---------------------------------------------------------------*)

//Try to reset the variable for connection on the GVL. When all is normal then the Lynus Mqtt connection function set this variable to true in the next cycle
//When we have no connection to the backend then after Lynus_Standards.Constants_General.tTimeDissableLynusFunctions days the Function is dissabled with all of his functionalities
timResetConnectionOnGVL(IN:= NOT timResetConnectionOnGVL.Q, PT:= T#1H, Q=> , ET=> );
	IF timResetConnectionOnGVL.Q THEN Lynus_Standards.GVL_Communicator.bStateConnectionToEnableFunctions := FALSE; END_IF
		IF NOT Lynus_Standards.GVL_Communicator.bStateConnectionToEnableFunctions THEN timDissableFunctions.IN := TRUE; ELSE timDissableFunctions.IN := FALSE; END_IF  
			timDissableFunctions(IN:= , PT:= Lynus_Standards.Constants_General.tTimeDissableLynusFunctions, Q=> , ET=> );
			
(*------------------------------------------------------------------------------------------State Machine Read---------------------------------------------------------------------------------------------*)

//When the function is not enabled then the fronius control by himself without modbus tcp connection
IF NOT bEnable OR timDissableFunctions.Q THEN bActivateControl := FALSE; END_IF

//Start the Statemachine
FPEnable(CLK:= bEnable, Q=> );
	FPActivateControl(CLK:= bActivateControl, Q=> );
		FNTimDissable(CLK:= timDissableFunctions.Q, Q=> );
			IF (FPEnable.Q AND iStateModbusRead = 0 AND iStateModbusRead = 0 AND iStateModbusError = 0) OR
				(bEnable AND FPActivateControl.Q AND iStateModbusRead = 0 AND iStateModbusRead = 0 AND iStateModbusError = 0) OR
					(bEnable AND FNTimDissable.Q AND iStateModbusRead = 0 AND iStateModbusRead = 0 AND iStateModbusError = 0) THEN 
						iStateModbusRead := 1; 
			END_IF
				IF NOT bEnable OR NOT bActivateControl THEN iStateModbusRead := 0; iStateModbusWrite := 0; iStateModbusError := 0; END_IF

//Timer for delay
timDelay(IN:= , PT:= T#500MS, Q=> , ET=> );

//Timer for Timeout in Statemachine
IF (iStateModbusRead > 0 AND iStateModbusRead <= 2 AND iStateModbusRead = iStateModbus_CP) OR
		(iStateModbusWrite > 0 AND iStateModbusWrite <= 1 AND iStateModbusWrite = iStateModbus_CP) THEN
			timTimeout.IN := TRUE;
ELSE	
			timTimeout.IN := FALSE;
END_IF 
	IF iStateModbusRead = 0 AND iStateModbusWrite = 0 THEN timTimeout.IN := FALSE; END_IF
		timTimeout(IN:= , PT:= T#20S, Q=> , ET=> );

CASE iStateModbusRead OF
	
	0://Init State
		iStateModbus_CP := 0;
			timDelay.IN := FALSE;
			
		stDataXelectrix.eBatteryState := E_Xelectrix_BatteryState.eNoDataReceived;
			stDataXelectrix.eGridState := E_Xelectrix_GridState.eNoDataReceived;
				stDataXelectrix.eOperatingState := E_Xelectrix_OperatingState.eNoDataReceived;	
					stDataXelectrix.bFunctionIsActive := FALSE;
			
		fbMBRead_FC3.bExecute := FALSE;
			fbMBWrite_FC16.bExecute := FALSE;	

	1://Read all the Data
		stDataXelectrix.bFunctionIsActive := TRUE;
			iStateModbus_CP := iStateModbusRead;
		
		//Reset Write
		fbMBWrite_FC16.bExecute := FALSE;
			arrBuffer_FC16[1] := 0; arrBuffer_FC16[2] := 0;
		
		//Start Read
		fbMBRead_FC3.nQuantity := 48;
			fbMBRead_FC3.nMBAddr := 0;
				fbMBRead_FC3.bExecute := TRUE;
			
		IF fbMBRead_FC3.bBusy THEN timDelay.IN := TRUE; END_IF
		
		//Wait for Delay, copy Data and then next step
		IF NOT fbMBRead_FC3.bBusy AND NOT fbMBRead_FC3.bError AND timDelay.Q THEN
			//Grid State
			IF arrBuffer_FC3[1] = 0 THEN stDataXelectrix.eGridState := E_Xelectrix_GridState.eOff; 
			ELSIF arrBuffer_FC3[1] = 1 THEN stDataXelectrix.eGridState := E_Xelectrix_GridState.eIslandMode;
			ELSIF arrBuffer_FC3[1] = 2 THEN stDataXelectrix.eGridState := E_Xelectrix_GridState.eOnline;
			ELSIF arrBuffer_FC3[1] = 3 THEN stDataXelectrix.eGridState := E_Xelectrix_GridState.eError;   	
			END_IF
			
			(*------------------------------------------Workaround why AC device deliver sometimes 0 Value--------------------------------------------------------*)
			byNumberOfZero := 0;
				FOR byLPWorkAroundACDevice := 6 TO 9 BY 1 DO
					IF arrBuffer_FC3[byLPWorkAroundACDevice] = 0 THEN byNumberOfZero := byNumberOfZero + 1; END_IF  
				END_FOR

			IF byNumberOfZero = 0 THEN
				//Real Power (Scale factor is * 100 for W)
				fbEMGrid.lrPowerTotal := INT_TO_LREAL(WORD_TO_INT(arrBuffer_FC3[2])) * 100;
				//Reactive Power (Scale factor is * 100 for var)
				fbEMGrid.lrReactivePowerTotal := INT_TO_LREAL(WORD_TO_INT(arrBuffer_FC3[3])) * 100; 
				//Frequency (Scale factor is / 100 for Hz)
				fbEMGrid.lrFrequency := INT_TO_LREAL(WORD_TO_INT(arrBuffer_FC3[6])) / 100;
				//Voltage L1/N (Scale factor is / 10 for V)
				fbEMGrid.lrVoltageL1N := INT_TO_LREAL(WORD_TO_INT(arrBuffer_FC3[7])) / 10;
				//Voltage L2/N (Scale factor is / 10 for V)
				fbEMGrid.lrVoltageL2N := INT_TO_LREAL(WORD_TO_INT(arrBuffer_FC3[8])) / 10;
				//Voltage L3/N (Scale factor is / 10 for V)
				fbEMGrid.lrVoltageL3N := INT_TO_LREAL(WORD_TO_INT(arrBuffer_FC3[9])) / 10;
				//Current L1 (Scale factor is * 100 for mA)
				fbEMGrid.lrCurrentL1 := INT_TO_LREAL(WORD_TO_INT(arrBuffer_FC3[10])) * 100;
					//Make / 1000 for A
					fbEMGrid.lrCurrentL1 := fbEMGrid.lrCurrentL1 / 1000;
				//Current L2 (Scale factor is * 100 for mA)
				fbEMGrid.lrCurrentL2 := INT_TO_LREAL(WORD_TO_INT(arrBuffer_FC3[11])) * 100;
					//Make / 1000 for A
					fbEMGrid.lrCurrentL2 := fbEMGrid.lrCurrentL2 / 1000;
				//Current L3 (Scale factor is * 100 for mA)
				fbEMGrid.lrCurrentL3 := INT_TO_LREAL(WORD_TO_INT(arrBuffer_FC3[12])) * 100;
					//Make / 1000 for A
					fbEMGrid.lrCurrentL3 := fbEMGrid.lrCurrentL3 / 1000;
			END_IF	
			(*-----------------------------------------------------------------------------------------------------------------------------------------------------*)
			
			//Max Charge Power (Scale factor is * 100 for W)
			fbBatteryInverter.rMaxChargePowerBattInverter := INT_TO_REAL(WORD_TO_INT(arrBuffer_FC3[14])) * 100; 
			//Max Discharge Power (Scale factor is * 100 for W)
			fbBatteryInverter.rMaxDischargePowerBattInverter := INT_TO_REAL(WORD_TO_INT(arrBuffer_FC3[15])) * 100;  
				
				//SOC (No Scalefactor. Is %)	
				fbBattery.dwBatterySOC := INT_TO_DWORD(WORD_TO_INT(arrBuffer_FC3[21]));
					fbBatteryInverter.dwBatterSOC := INT_TO_DWORD(WORD_TO_INT(arrBuffer_FC3[21]));
				//Battery Temperature (Scale factor is / 100 for °C)
				fbBattery.lrBatteryTemp := INT_TO_LREAL(WORD_TO_INT(arrBuffer_FC3[23])) / 100; 
				//Battery State
				IF arrBuffer_FC3[24] = 0 THEN stDataXelectrix.eBatteryState := E_Xelectrix_BatteryState.eOff;
				ELSIF arrBuffer_FC3[24] = 1 THEN stDataXelectrix.eBatteryState := E_Xelectrix_BatteryState.eStartUp;
				ELSIF arrBuffer_FC3[24] = 2 THEN stDataXelectrix.eBatteryState := E_Xelectrix_BatteryState.eBalancing;
				ELSIF arrBuffer_FC3[24] = 3 THEN stDataXelectrix.eBatteryState := E_Xelectrix_BatteryState.eReady;
				ELSIF arrBuffer_FC3[24] = 4 THEN stDataXelectrix.eBatteryState := E_Xelectrix_BatteryState.eOperating;
				ELSIF arrBuffer_FC3[24] = 6 THEN stDataXelectrix.eBatteryState := E_Xelectrix_BatteryState.eError;
				END_IF  
				//Operating State
				IF arrBuffer_FC3[25] = 0 THEN stDataXelectrix.eOperatingState := E_Xelectrix_OperatingState.eOff;
				ELSIF arrBuffer_FC3[25] = 1 THEN stDataXelectrix.eOperatingState := E_Xelectrix_OperatingState.eDischarge;
				ELSIF arrBuffer_FC3[25] = 2 THEN stDataXelectrix.eOperatingState := E_Xelectrix_OperatingState.eCharge;
				ELSIF arrBuffer_FC3[25] = 3 THEN stDataXelectrix.eOperatingState := E_Xelectrix_OperatingState.eIdle;
				END_IF
				//Battery Capacity in Wh (Scale factor is * 100 for Wh), but make the calculation for kWh
				lrMaxCapacityBattery_OUT := arrBuffer_FC3[26] * 100;
					lrMaxCapacityBattery_OUT := lrMaxCapacityBattery_OUT / 1000;
				//Battery Current (Scale factor is * 100 for mA)
				fbBattery.lrBatteryCurrent := INT_TO_LREAL(WORD_TO_INT(arrBuffer_FC3[27])) * 100;
					//Make / 1000 for A
					fbBattery.lrBatteryCurrent := fbBattery.lrBatteryCurrent / 1000;
						//Change the sign because in view from the Battery - is discharge and + is charge. But we use vice versa	
						fbBattery.lrBatteryCurrent := fbBattery.lrBatteryCurrent * - 1; 
				//Battery Voltage 
				fbBattery.rBatteryVoltage := INT_TO_REAL(WORD_TO_INT(arrBuffer_FC3[28]));
				//Max Charge Current (Scale factor is * 100 for mA)
				fbBattery.rMaxDcChargeCurrentBattery := INT_TO_REAL(WORD_TO_INT(arrBuffer_FC3[29])) * 100; 
					//Make / 1000 for A
					fbBattery.rMaxDcChargeCurrentBattery := fbBattery.rMaxDcChargeCurrentBattery / 1000;
				//Max Discharge Current (Scale factor is * 100 for mA)
				//Its allways a negative raw value
				iMaxDcDischargeCurrentBattery := WORD_TO_INT(arrBuffer_FC3[30]);
					iMaxDcDischargeCurrentBattery := iMaxDcDischargeCurrentBattery * - 1;
						fbBattery.rMaxDcDischargeCurrentBattery := INT_TO_REAL(iMaxDcDischargeCurrentBattery) * 100; 
					//Make / 1000 for A
					fbBattery.rMaxDcDischargeCurrentBattery := fbBattery.rMaxDcDischargeCurrentBattery / 1000;
					
